FUNCTION_BLOCK "FB_Robot"
{ S7_Optimized_Access := 'TRUE' }
VERSION : 0.1
   VAR
      cmdStatus { S7_SetPoint := 'False'} : "UDT_CMD";
   END_VAR
   VAR RETAIN
      Dispatcher : Array[0..31] of Int;
   END_VAR
   VAR
      Auto : Bool;
      RemoteMode : Bool := TRUE;
      Status : Int;
      oldStatus { ExternalAccessible := 'False'; ExternalVisible := 'False'; ExternalWritable := 'False'} : Int;
      workCondition : Int;   // Status REMOTE, LOCAL, MANUAL
   END_VAR
   VAR RETAIN
      communication_OK : Bool;   // Communication with robot's brain OK
   END_VAR
   VAR
      MissionCode : Int;
      BoxRequested : Int := 1;   // Which warehouse used for mission
      GripperRequested : Int;
      MCRequested : Int;
      PalletRequested : Int;
      Tray_ID : Int;
      Error : Int;   // Every error raised during the cycle
      timeoutLifeBit {InstructionName := 'TON_TIME'; LibVersion := '1.0'; S7_SetPoint := 'False'} : TON_TIME;
   END_VAR
   VAR RETAIN
      Gripper_ID : Array[1..2] of Int;   // Codes of gripper mounted
      GripperOccuped : Array[1..2] of Bool;   // Gripper occuped status
   END_VAR
   VAR
      queryTemp : String;
      paramsTemp { ExternalAccessible := 'False'; ExternalVisible := 'False'; ExternalWritable := 'False'} : Array[0..5] of Int;
      queryStartExecution { ExternalAccessible := 'False'; ExternalVisible := 'False'; ExternalWritable := 'False'} : Bool;
      PollingDB {InstructionName := 'TON_TIME'; LibVersion := '1.0'; S7_SetPoint := 'False'} : Array[1..5] of TON_TIME;
      lastMission { S7_SetPoint := 'True'} : Int;
      WAIT_END_MISSION : Bool;
      HOLD : Bool;
      PalletPosition : Int;
      checkInconsistenceFailed : Bool;
      speedRequest : Int;
      tonCoerenza {InstructionName := 'TON_TIME'; LibVersion := '1.0'; S7_SetPoint := 'False'} : TON_TIME;
      auxOK_old { S7_SetPoint := 'True'} : Bool;
      swapDataReady : Bool;
      tonSwapA {InstructionName := 'TON_TIME'; LibVersion := '1.0'; S7_SetPoint := 'False'} : TON_TIME;
      tonSwapB {InstructionName := 'TON_TIME'; LibVersion := '1.0'} : TON_TIME;
      currentGripperHasHook { S7_SetPoint := 'True'} : Bool;
      PartSubPos : Int;
      declGripper : Int;
      declCont1 : Int;
      declId1 : Int;
      declCont2 : Int;
      declId2 : Int;
      declMap : Int;
      mounted_old : Int := -1;
      closed1_old : Int := -1;
      tonSafetyPub {InstructionName := 'TON_TIME'; LibVersion := '1.0'; S7_SetPoint := 'False'} : TON_TIME;
      zPlaceTemp { S7_SetPoint := 'True'} : DInt;
      PartSubPosMC : Int;
      TrayIdMC : Int;
      xPushTemp : DInt;
      xStopTemp : DInt;
      xPushOffsetMC : DInt;
      xPlaceTemp : DInt;
      declSubPos : Int;
      declStato : Int;
      declTipo : Int;
      retryPick : Bool;
      tonExtract {InstructionName := 'TON_TIME'; LibVersion := '1.0'; S7_SetPoint := 'False'} : TON_TIME;
      OrderIdMC { S7_SetPoint := 'True'} : Int;
      holdButton : Bool;
   END_VAR

   VAR_TEMP
      pieceReq : Int;
      Dispatcher_old : Array[0..31] of Int;
      i : Int;
      RESET_ALL_DISPATCH : Bool;
      temp : Int;
      robotInPendant : Bool;
   END_VAR


BEGIN
	(* Implementato dentro alla classe del Robot
	REGION LIFE BIT
	    "DB_RobotMission".SystemSignals_IN.LIFEBIT_IN := NOT "DB_RobotMissionStatus".systemsignals.LIFE_BIT;

	    #timeoutLifeBit(IN := "DB_RobotMission".SystemSignals_IN.LIFEBIT_IN <> "DB_RobotMissionStatus".systemsignals.LIFE_BIT,
	                    PT := T#3S);

	    IF (#timeoutLifeBit.Q) THEN
	        //salva su DB errore di comunicazione con robot
	        #communication_OK := FALSE;
	    END_IF;
	END_REGION
	*)
	// Il flag va abbassato SOLO quando la query e' entrata davvero nel ponte.
	// Senza il controllo di lunghezza, due stringhe vuote si confermano a vicenda
	// e il flag cade su una query mai partita: la catena resta appesa per sempre
	// (visto 4/9 sulla missione 16, errore 13599 in loop).
	IF LEN(#queryTemp) > 0
	    AND #queryTemp = "SqlCommands".sqlCommands[0]
	    AND #queryStartExecution
	THEN
	    #queryStartExecution := FALSE;
	END_IF;

	REGION Status

	    #Status := DINT_TO_INT("AUTO");
	    IF NOT #HOLD AND ("DB_RobotMissionStatus".StatusCode = "cmd_acquired" OR
	        "DB_RobotMissionStatus".StatusCode = "cmd_executing") THEN
	        #Status := DINT_TO_INT("WORKING");
	    ELSIF NOT #HOLD AND ("DB_RobotMissionStatus".StatusCode = "cmd_aborted" OR
	        "DB_RobotMissionStatus".StatusCode = "cmd_rejected") THEN
	        #Status := DINT_TO_INT("ABORTED");
	    ELSIF NOT #HOLD AND (#Dispatcher["_master"] = 9999 OR
	        #Error <> 0 OR
	        "DB_RobotMissionStatus".StatusRegister.Alarm) THEN
	        #Status := DINT_TO_INT("ALARM");
	    ELSIF NOT #communication_OK THEN
	        #Status := DINT_TO_INT("NOT_DEFINED");
	    ELSIF NOT #HOLD AND NOT "DB_RobotMissionStatus".StatusRegister.Executing AND #Auto THEN
	        #Status := DINT_TO_INT("OFF");
	    ELSIF #HOLD THEN
	        #Status := DINT_TO_INT("HOLD");
	    ELSIF NOT #Auto THEN
	        #Status := DINT_TO_INT("MANUAL");
	    ELSE
	        #Status := DINT_TO_INT("REMOTE");
	    END_IF;

	    IF (#Status <> #oldStatus AND #Status >= 0) THEN
	        IF "DB_RobotMissionStatus".StatusRegister.Alarm THEN
	            "FC_MQTT"(insert := true,
	                      send := false,
	                      topic := 'FROM_PLANT/DESCR/ROBOT',
	                      payload := STRING_TO_WSTRING("INT_TO_STRING_WITHOUT_SIGN"("Alarmcode")));
	        ELSE
	            "FC_MQTT"(insert := true,
	                      "send" := false,
	                      topic := 'FROM_PLANT/DESCR/ROBOT',
	                      payload := STRING_TO_WSTRING("INT_TO_STRING_WITHOUT_SIGN"(#Error)));
	        END_IF;
	        "FC_MQTT"(insert := true,
	                  send := false,
	                  topic := 'FROM_PLANT/STATUS/ROBOT',
	                  payload := STRING_TO_WSTRING("INT_TO_STRING_WITHOUT_SIGN"(#Status)));
	        #oldStatus := #Status;
	    END_IF;

	    //controllo ad ogni ciclo
	    #Status := DINT_TO_INT("REMOTE");

	    IF (#Status <> #workCondition AND #Status >= 0) THEN
	        "FC_MQTT"(insert := true,
	                  send := false,
	                  topic := 'FROM_PLANT/STATUS/ROBOT',
	                  payload := STRING_TO_WSTRING("INT_TO_STRING_WITHOUT_SIGN"(#Status)));
	        #workCondition := #Status;
	    END_IF;
	END_REGION ;

	FOR #i := 0 TO 31 DO
	    #Dispatcher_old[#i] := #Dispatcher[#i];
	END_FOR;

	REGION Manager CMD from HMI
	    // Modo cella: DB_Robot.RemoteMode (TRUE = automatico, FALSE = manuale/locale).
	    // Scritto SOLO qui dai comandi 81/82 — il robot non partecipa al giro modalita'.
	    // Robot sotto pendant (manuale suo): nessun comando di movimento accettato.
	    #robotInPendant := "sys_manual_T1" OR "sys_manual_Full";
	    #RemoteMode := NOT #HOLD;   // modo cella derivato: HOLD = manuale

	    // ---- Comandi accettati in ogni condizione ----
	    IF "DB_MQTT".lastTopicReceived = 'ROBOT' THEN
	        CASE "DB_MQTT".lastCmdReceived OF
	            "CMD_HOLD":
	                // IL PULSANTE E' MASTER (19/9): un hold messo col pulsante fisico
	                // lo toglie solo il pulsante. Dal pannello si puo' mettere
	                // l'hold e togliere il proprio, non quello di chi sta in campo
	                // davanti alla cella. La gerarchia la tiene FB5, che scrive
	                // holdButton: qui si legge e basta.
	                IF NOT #holdButton THEN
	                    #HOLD := NOT #HOLD;
	                END_IF;
	            "CMD_changeRobotSpeed":
	                #speedRequest := "DB_MQTT".lastParams[0];
	            "CMD_Refresh":  // 90: ripubblica tutti gli one-shot
	                #oldStatus := -1;
	                #lastMission := -1;
	                #auxOK_old := NOT "Main_Safety_RTG1_DB".Aux_OK;
	                #mounted_old := -1;
	                #closed1_old := -1;
	                "DB_MC1".brandID_req_old := -1;
	                "DB_MC1".brandID_act_old := -1;
	                "DB_MC1".declPallet_old := -1;
	                "DB_MC1".declPiece_old := -1;
	                "DB_MC1".declVice_old := -1;
	                FOR #i := 0 TO 31 DO
	                    #Dispatcher_old[#i] := -1;
	                END_FOR;
	                "DB_MQTT".lastCmdReceived := 0;
	        END_CASE;
	    END_IF;

	    // ---- Restart main program: solo con orchestrazione in HOLD ----
	    IF "DB_MQTT".lastTopicReceived = 'ROBOT' AND #HOLD THEN
	        CASE "DB_MQTT".lastCmdReceived OF
	            "CMD_RestartMainProg":
	                "DB_RobotMission".Command := "CMD_RestartMainProg";
	                "DB_MQTT".lastCmdReceived := 0;
	                #WAIT_END_MISSION := FALSE;
	                // il restart del programma robot abbandona la missione in corso (5/10):
	                // si azzerano le catene come per i movimenti manuali, altrimenti
	                // restano ad aspettare un "eseguito" che non arrivera' mai.
	                #RESET_ALL_DISPATCH := TRUE;
	                #MissionCode := 0;
	        END_CASE;
	    END_IF;

	    // ---- Canale libero: modo cella + reset, validi in ENTRAMBI i modi ----
	    IF "DB_MQTT".lastTopicReceived = 'ROBOT'
	        AND "DB_RobotMissionStatus".StatusCode <> "cmd_acquired"
	        AND "DB_RobotMissionStatus".StatusCode <> "cmd_executing"
	    THEN
	        CASE "DB_MQTT".lastCmdReceived OF
	            "CMD_RobotReset":
	                #Error := 0;
	                "DB_RobotMission".Command := "CMD_RobotReset"; //arriva direttamente nella missione robot
	                #MissionCode := 0;
	                #RESET_ALL_DISPATCH := TRUE;
	                #WAIT_END_MISSION := TRUE;

	                // IL RESET DEVE FERMARE ANCHE L'ORCHESTRAZIONE MACCHINA (16/9).
	                // Prima azzerava solo le catene di FB7: FB204 restava dov'era e
	                // riprendeva da uno stato che non esisteva piu'. Visto in campo:
	                // reset a meta' deposito del finito -> il 95 substate 1 vede
	                // MissionCode = 0 (appena azzerato QUI) e conclude che lo scarico
	                // e' finito, prosegue sui registri di bordo troncati, e arriva a
	                // rilanciare la RICETTA su un pezzo GIA' LAVORATO ancora in morsa.
	                "DB_MC1".Dispatcher["_master"] := 0;
	                "DB_MC2".Dispatcher["_master"] := 0;

	                "DB_MQTT".lastCmdReceived := 0;
	        END_CASE;

	        // ---- Comandi manuali: SOLO cella in locale E robot non in pendant ----
	        IF NOT #RemoteMode AND NOT #robotInPendant THEN
	            CASE "DB_MQTT".lastCmdReceived OF
	                "CMD_RobotToHomePos":
	                    "DB_RobotMission".Command := "CMD_RobotToHomePos";
	                    "DB_MQTT".lastCmdReceived := 0;
	                    #WAIT_END_MISSION := TRUE;
	                    #RESET_ALL_DISPATCH := TRUE; // abort missioni pendenti: no falso latch da 3 del movimento manuale
	                    #MissionCode := 0;
	                "CMD_RobotMaintenancePos":
	                    "DB_RobotMission".Command := "CMD_RobotMaintenancePos";
	                    "DB_MQTT".lastCmdReceived := 0;
	                    #WAIT_END_MISSION := TRUE;
	                    #RESET_ALL_DISPATCH := TRUE; // abort missioni pendenti: no falso latch da 3 del movimento manuale
	                    #MissionCode := 0;
	                "CMD_RobotPositioning":
	                    "DB_RobotMission".Command := "CMD_RobotPositioning"; // riceve comandi del tipo 15;1
	                    "DB_RobotMission".Unit_code := "DB_MQTT".lastParams[0];
	                    "DB_MQTT".lastCmdReceived := 0;
	                    #WAIT_END_MISSION := TRUE;
	                    #RESET_ALL_DISPATCH := TRUE; // abort missioni pendenti: no falso latch da 3 del movimento manuale
	                    #MissionCode := 0;
	                "CMD_RobotPositioning_BOX1":
	                    "DB_RobotMission".Command := "CMD_RobotPositioning";
	                    "DB_RobotMission".Unit_code := "Warehouse1";
	                    "DB_MQTT".lastCmdReceived := 0;
	                    #WAIT_END_MISSION := TRUE;
	                    #RESET_ALL_DISPATCH := TRUE; // abort missioni pendenti: no falso latch da 3 del movimento manuale
	                    #MissionCode := 0;
	                "CMD_RobotPositioning_MC1":
	                    "DB_RobotMission".Command := "CMD_RobotPositioning";
	                    "DB_RobotMission".Unit_code := "MC1";
	                    "DB_MQTT".lastCmdReceived := 0;
	                    #WAIT_END_MISSION := TRUE;
	                    #RESET_ALL_DISPATCH := TRUE; // abort missioni pendenti: no falso latch da 3 del movimento manuale
	                    #MissionCode := 0;
	                "CMD_RobotPickGripper":
	                    "DB_MQTT".lastCmdReceived := 0;
	                    #MissionCode := "MISSION_LoadGripper";
	                    #GripperRequested := "DB_MQTT".lastParams[0];
	                    #WAIT_END_MISSION := TRUE;
	                "CMD_RobotRemoveGripper":
	                    "DB_MQTT".lastCmdReceived := 0;
	                    #MissionCode := "MISSION_UnloadGripper";
	                    #WAIT_END_MISSION := TRUE;
	                "CMD_RobotExtractTray":
	                    #Tray_ID := DINT_TO_INT("DB_MQTT".lastParams[0]);  // <-- riga nuova
	                    #MissionCode := "MISSION_ExtractTray";
	                    "DB_MQTT".lastCmdReceived := 0;
	                    #WAIT_END_MISSION := TRUE;
	                "CMD_RobotReleaseTray":
	                    #MissionCode := "MISSION_ReleaseTray";
	                    "DB_MQTT".lastCmdReceived := 0;
	                    #WAIT_END_MISSION := TRUE;
	                "CMD_RobotPickObject":
	                    "DB_RobotMission".Object_Type := "DB_MQTT".lastParams[0];
	                    #PalletRequested := "DB_MQTT".lastParams[1];
	                    CASE "DB_RobotMission".Object_Type OF
	                        "Pallet":
	                            #PalletPosition := "DB_MQTT".lastParams[2];
	                            IF #PalletPosition = 0 THEN
	                                #MissionCode := "MISSION_PickPallet_MC_HMI";
	                                #MCRequested := 1;
	                            ELSE
	                                #MissionCode := "MISSION_Load_Pallet";
	                                #MCRequested := 0;
	                            END_IF;
	                            "DB_MQTT".lastCmdReceived := 0;
	                            #WAIT_END_MISSION := TRUE;
	                        "Part": //TODO
	                            ;
	                        "ViceWithoutPart":
	                            ;
	                        "ViceWithPart":
	                            ;
	                    END_CASE;
	                "CMD_RobotPlaceObject":
	                    "DB_RobotMission".Object_Type := "DB_MQTT".lastParams[0];
	                    #PalletRequested := "DB_MQTT".lastParams[1];
	                    CASE "DB_RobotMission".Object_Type OF
	                        "Pallet":
	                            #PalletPosition := "DB_MQTT".lastParams[2];
	                            IF #PalletPosition = 0 THEN
	                                #MissionCode := "MISSION_PlacePallet_MC_HMI";
	                                #MCRequested := 1;
	                            ELSE
	                                #MissionCode := "MISSION_Unload_Pallet";
	                                #MCRequested := 0;
	                            END_IF;
	                            "DB_MQTT".lastCmdReceived := 0;
	                            #WAIT_END_MISSION := TRUE;
	                        "Part": //TODO
	                            ;
	                        "ViceWithoutPart":
	                            ;
	                        "ViceWithPart":
	                            ;
	                    END_CASE;
	                "CMD_HMI_SwapGripper":
	                    "DB_MQTT".lastCmdReceived := 0;
	                    #GripperRequested := "DB_MQTT".lastParams[0];
	                    #MissionCode := "MISSION_SwapGripper";
	                    #WAIT_END_MISSION := TRUE;

	                "CMD_DeclarePosition_TRAY":   // 39;subpos;stato  (2 vuota, 4 grezzo, 5 finito)
	                    #declSubPos := DINT_TO_INT("DB_MQTT".lastParams[0]);
	                    #declStato := DINT_TO_INT("DB_MQTT".lastParams[1]);
	                    #declTipo := 0;                         // ramo STATO, non TIPO
	                    IF "DB_BOX_1".ExtractedTray <= 0 THEN
	                        #Error := 20001;                    // nessun cassetto estratto
	                    ELSIF #declSubPos <= 0 THEN
	                        #Error := 20002;                    // posizione non valida
	                    ELSIF #declStato <> 2 AND #declStato <> 4 AND #declStato <> 5 THEN
	                        #Error := 20005;                    // stato non ammesso
	                    ELSE
	                        #Dispatcher["_Declare_Position"] := 10;
	                    END_IF;
	                    "DB_MQTT".lastCmdReceived := 0;
	                    #WAIT_END_MISSION := FALSE;   // nessun movimento robot

	                "CMD_DeclarePieceType_TRAY":   // 44;partType  tipo pezzo dell'INTERO cassetto estratto
	                    #declTipo := DINT_TO_INT("DB_MQTT".lastParams[0]);
	                    IF "DB_BOX_1".ExtractedTray <= 0 THEN
	                        #Error := 20001;                    // nessun cassetto estratto
	                    ELSIF #declTipo <= 0 THEN
	                        #Error := 20008;                    // tipo pezzo non valido
	                    ELSE
	                        #Dispatcher["_Declare_Position"] := 15;   // ramo TIPO
	                    END_IF;
	                    "DB_MQTT".lastCmdReceived := 0;
	                    #WAIT_END_MISSION := FALSE;   // nessun movimento robot

	                "CMD_RobotPickPartTray":   // 27;subpos;gripperID  (gripperID 0 = pinza a bordo)
	                    IF "DB_BOX_1".ExtractedTray <= 0 THEN
	                        #Error := 20001;                    // nessun cassetto estratto
	                    ELSIF DINT_TO_INT("DB_MQTT".lastParams[0]) <= 0 THEN
	                        #Error := 20002;                    // posizione pezzo non valida
	                    ELSIF DINT_TO_INT("DB_MQTT".lastParams[1]) = 0 AND #Gripper_ID[1] = 0 THEN
	                        #Error := 22;                       // flangia vuota e nessuna pinza richiesta
	                    ELSE
	                        #PartSubPos := DINT_TO_INT("DB_MQTT".lastParams[0]);
	                        #GripperRequested := DINT_TO_INT("DB_MQTT".lastParams[1]);
	                        IF #GripperRequested = 0 THEN
	                            #GripperRequested := #Gripper_ID[1];
	                        END_IF;
	                        #Tray_ID := "DB_BOX_1".ExtractedTray;
	                        #MCRequested := 0;
	                        #MissionCode := "MISSION_PickPart_TRAY_HMI";
	                        #WAIT_END_MISSION := TRUE;
	                    END_IF;
	                    "DB_MQTT".lastCmdReceived := 0;

	                "CMD_RobotPlacePartTray":  // 28;subpos  (0 = prima posizione vuota)
	                    IF "DB_BOX_1".ExtractedTray <= 0 THEN
	                        #Error := 20001;
	                    ELSE
	                        #PartSubPos := DINT_TO_INT("DB_MQTT".lastParams[0]);
	                        #Tray_ID := "DB_BOX_1".ExtractedTray;
	                        #MCRequested := 0;
	                        #MissionCode := "MISSION_PlacePart_TRAY_HMI";
	                        #WAIT_END_MISSION := TRUE;
	                    END_IF;
	                    "DB_MQTT".lastCmdReceived := 0;

	                "CMD_RobotPickPartMC":     // 29;gripperID  (0 = pinza a bordo)
	                    IF DINT_TO_INT("DB_MQTT".lastParams[0]) = 0 AND #Gripper_ID[1] = 0 THEN
	                        #Error := 22;
	                    ELSE
	                        #GripperRequested := DINT_TO_INT("DB_MQTT".lastParams[0]);
	                        IF #GripperRequested = 0 THEN
	                            #GripperRequested := #Gripper_ID[1];
	                        END_IF;
	                        #MCRequested := 1;                  // MC2 non esiste in questa cella
	                        #MissionCode := "MISSION_PickPart_MC_HMI";
	                        #WAIT_END_MISSION := TRUE;
	                    END_IF;
	                    "DB_MQTT".lastCmdReceived := 0;

	                "CMD_RobotPlacePartMC":    // 30  (pezzo a bordo -> morsa MC1)
	                    #MCRequested := 1;
	                    #GripperRequested := #Gripper_ID[1];
	                    #MissionCode := "MISSION_PlacePart_MC_HMI";
	                    #WAIT_END_MISSION := TRUE;
	                    "DB_MQTT".lastCmdReceived := 0;
	                "CMD_RobotPickPlacePartMC":  // 244  (finito da morsa + grezzo in morsa, un ingresso)
	                    IF NOT #GripperOccuped[1] THEN
	                        #Error := 20003;                    // nessun grezzo a bordo lato 1
	                    ELSIF #GripperOccuped[2] THEN
	                        #Error := 20004;                    // lato finito gia' occupato
	                    ELSE
	                        #MCRequested := 1;
	                        #GripperRequested := #Gripper_ID[1];
	                        #MissionCode := "MISSION_PickPlacePart_MC";
	                        #WAIT_END_MISSION := TRUE;
	                    END_IF;
	                    "DB_MQTT".lastCmdReceived := 0;
	                "CMD_OpenGripper1":
	                    "DB_MQTT".lastCmdReceived := 0;
	                    #MissionCode := "MISSION_OpenGripper1";
	                    #WAIT_END_MISSION := TRUE;
	                "CMD_CloseGripper1":
	                    "DB_MQTT".lastCmdReceived := 0;
	                    #MissionCode := "MISSION_CloseGripper1";
	                    #WAIT_END_MISSION := TRUE;
	                "CMD_OpenGripper2":
	                    IF #Gripper_ID[2] = 0 THEN
	                        #Error := 944;   // lato 2 inesistente sulla pinza a bordo
	                    ELSE
	                        #MissionCode := "MISSION_OpenGripper2";
	                        #WAIT_END_MISSION := TRUE;
	                    END_IF;
	                    "DB_MQTT".lastCmdReceived := 0;
	                "CMD_CloseGripper2":
	                    IF #Gripper_ID[2] = 0 THEN
	                        #Error := 944;
	                    ELSE
	                        #MissionCode := "MISSION_CloseGripper2";
	                        #WAIT_END_MISSION := TRUE;
	                    END_IF;
	                    "DB_MQTT".lastCmdReceived := 0;
	                "CMD_RobotDeclareState":   // 35;gripperID;cont1;id1;cont2;id2  (cont: 0=vuoto 1=grezzo 2=finito 3=pallet)
	                    #declGripper := DINT_TO_INT("DB_MQTT".lastParams[0]);
	                    #declCont1 := DINT_TO_INT("DB_MQTT".lastParams[1]);
	                    #declId1 := DINT_TO_INT("DB_MQTT".lastParams[2]);
	                    #declCont2 := DINT_TO_INT("DB_MQTT".lastParams[3]);
	                    #declId2 := DINT_TO_INT("DB_MQTT".lastParams[4]);
	                    #Error := 0;
	                    #MissionCode := 0;
	                    #Dispatcher["_Declare_State"] := 10;
	                    "DB_MQTT".lastCmdReceived := 0;
	                    #WAIT_END_MISSION := FALSE;   // nessun movimento robot
	            END_CASE;
	        END_IF;
	    END_IF;

	    // ---- Completamento comando (invariato) ----
	    IF #WAIT_END_MISSION THEN
	        IF "DB_RobotMissionStatus".StatusCode = "cmd_executed" THEN
	            #WAIT_END_MISSION := FALSE;
	            //sync with robot
	            "DB_RobotMission".Command := 0;
	        ELSIF "DB_RobotMissionStatus".StatusCode = "cmd_rejected" OR "DB_RobotMissionStatus".StatusCode = "cmd_aborted" THEN
	            #WAIT_END_MISSION := FALSE;
	            // COMANDO MANUALE RIFIUTATO O ABORTITO (5/10): senza missione in
	            // corso si azzera anche il comando. Altrimenti il 4/5 resta esposto
	            // e la sorveglianza qui sotto lo attribuirebbe alla missione dopo.
	            IF #Dispatcher["_master"] = 0 THEN
	                "DB_RobotMission".Command := 0;
	            END_IF;
	        END_IF;
	    END_IF;

	    // ---- Sorveglianza risposta robot (5/10) ----
	    // Le risposte 4 (abortito) e 5 (rifiutato) erano gestite solo qui sopra,
	    // per i comandi manuali, e nelle catene chele. Le catene pezzi e cassetto
	    // restavano ad aspettare un 3 che non arriva: cella ferma con Error = 0 e
	    // nessuna spiegazione. Con una missione in corso e un comando al robot,
	    // una risposta anomala che dura 1 s diventa un errore dichiarato, che il
	    // reset (99) toglie. Il secondo di filtro evita di leggere lo StatusCode
	    // rimasto dal comando precedente nei primi cicli dopo un comando nuovo.
	    // Esclusi: lo scan del reset (99, AUX, ResetAreaRobot), in cui il master
	    // e' ancora valorizzato; l'HOLD, in cui il programma robot e' in pausa; la
	    // ripartenza del programma dopo HOLD o restart (FB8 dispatcher 0 e 1), che
	    // puo' durare fino a 17 s.
	    // Il codice 6 ("interrotto") NON e' gestito: non e' fra le costanti cmd_
	    // e va prima confermato col robotista.
	    // PollingDB[1] e' un timer gia' dichiarato e mai usato: nessuna variabile
	    // nuova, interfaccia invariata.
	    #PollingDB[1](IN := #Dispatcher["_master"] <> 0
	                  AND #Error = 0
	                  AND "DB_RobotMission".Command <> 0
	                  AND NOT #HOLD
	                  AND NOT #RESET_ALL_DISPATCH
	                  AND NOT "Start_AUX"
	                  AND NOT "ResetAreaRobot"
	                  AND "DB_Robot_Efort".dispatcher[0] = 0
	                  AND "DB_Robot_Efort".dispatcher[1] = 0
	                  AND ("DB_RobotMissionStatus".StatusCode = "cmd_aborted"
	                  OR "DB_RobotMissionStatus".StatusCode = "cmd_rejected"),
	                  PT := T#1s);
	    IF #PollingDB[1].Q THEN
	        IF "DB_RobotMissionStatus".StatusCode = "cmd_aborted" THEN
	            #Error := 961;   // missione abortita dal robot
	        ELSE
	            #Error := 962;   // comando rifiutato dal robot
	        END_IF;
	    END_IF;
	END_REGION

	REGION Cycle MASTER ROBOT

	    //DA TESTARE
	    (*IF "DB_RobotMissionStatus".StatusCode = "cmd_executed" THEN
	        "DB_RobotMission".Command := 0;
	    END_IF;
	    *)

	    IF NOT "Main_Safety_RTG1_DB".Aux_OK THEN
	        #MissionCode := 0;
	    END_IF;

	    #tonSwapA(IN := #Dispatcher["_master"] >= 973 AND #Dispatcher["_master"] <= 974,
	              PT := T#60s);
	    // TIMEOUT ESTESO AL 9781 (17/9): il 978 ora chiude in un ciclo e passa la
	    // registrazione alla catena unica. Senza estendere la sorveglianza, un ponte
	    // SQL occupato lascerebbe il master appeso al 9781 in silenzio, con la pinza
	    // gia' a bordo.
	    #tonSwapB(IN := #Dispatcher["_master"] = 978 OR #Dispatcher["_master"] = 9781,
	              PT := T#60s);
	    IF (#tonSwapA.Q OR #tonSwapB.Q) AND #Error = 0 THEN
	        #Error := 943;  // swap: timeout di fase (deposito o prelievo)
	    END_IF;

	    // SORVEGLIANZA CATENA CASSETTO (18/9): e' la terza catena che si pianta in
	    // silenzio. Il 12 aveva un ramo mancante — corretto — ma il principio resta:
	    // una catena senza timeout, quando si ferma, ferma anche il 750 che la
	    // aspetta e il 58 di FB204 che aspetta il 750, e nessuno lo dice.
	    // Tre minuti coprono estrazione e rilascio con margine largo.
	    #tonExtract(IN := #Dispatcher["Extract_TRAY"] > 0 OR #Dispatcher["Release_TRAY"] > 0,
	                PT := T#180s);
	    IF #tonExtract.Q AND #Error = 0 THEN
	        #Error := 19003;   // catena cassetto: timeout
	    END_IF;

	    IF #communication_OK THEN
	        CASE #Dispatcher["_master"] OF
	            0:
	                CASE #MissionCode OF
	                    "MISSION_LoadPallet_MC":        // pallet: Robot -> MC
	                        IF #RemoteMode AND
	                            "DB_RobotMissionStatus".StatusCode = "cmd_waitingNewCmd"
	                        THEN
	                            IF #MCRequested = 1 THEN
	                                IF "DB_MC1".order.GRIPPER4PALLET > 0 THEN
	                                    #GripperRequested := DINT_TO_INT("DB_MC1".order.GRIPPER4PALLET);
	                                    #Dispatcher["_master"] := 100;
	                                END_IF;
	                            ELSIF #MCRequested = 2 THEN
	                                IF "DB_MC1".order.GRIPPER4PALLET > 0 THEN
	                                    #GripperRequested := DINT_TO_INT("DB_MC2".order.GRIPPER4PALLET);
	                                    #Dispatcher["_master"] := 100;
	                                END_IF;
	                            ELSE
	                                #Dispatcher["_master"] := 0;
	                            END_IF;
	                        END_IF;
	                    "MISSION_UnloadPallet_MC":      // pallet: MC -> Robot
	                        IF #RemoteMode AND
	                            "DB_RobotMissionStatus".StatusCode = "cmd_waitingNewCmd"
	                        THEN
	                            IF #MCRequested = 1 THEN
	                                #GripperRequested := DINT_TO_INT("DB_MC1".order.GRIPPER4PALLET);
	                            ELSE
	                                #GripperRequested := DINT_TO_INT("DB_MC2".order.GRIPPER4PALLET);
	                            END_IF;
	                            #Dispatcher["_master"] := 200;
	                        END_IF;
	                    "MISSION_LoadPart_MC":          // part: Robot -> MC
	                        IF #RemoteMode AND
	                            "DB_RobotMissionStatus".StatusCode = "cmd_waitingNewCmd"
	                        THEN
	                            IF #MCRequested = 1 THEN
	                                #GripperRequested := DINT_TO_INT("DB_MC1".order.GRIPPER);
	                            ELSE
	                                #GripperRequested := DINT_TO_INT("DB_MC2".order.GRIPPER);
	                            END_IF;
	                            IF #GripperRequested > 0 THEN
	                                #Dispatcher["_master"] := 300;
	                            ELSE
	                                #Error := "MISSION_LoadPart_MC" * 100 + 10;  //Error 12010
	                            END_IF;
	                        END_IF;
	                    "MISSION_UnloadPart_MC":        // part: MC -> Robot
	                        IF #RemoteMode AND
	                            "DB_RobotMissionStatus".StatusCode = "cmd_waitingNewCmd"
	                        THEN
	                            IF #MCRequested = 1 THEN
	                                #GripperRequested := DINT_TO_INT("DB_MC1".order.GRIPPER);
	                            ELSE
	                                #GripperRequested := DINT_TO_INT("DB_MC2".order.GRIPPER);
	                            END_IF;
	                            IF #GripperRequested > 0 THEN
	                                #Dispatcher["_master"] := 400;
	                            ELSE
	                                #Error := "MISSION_UnloadPart_MC" * 100 + 10;  //Error 13010
	                            END_IF;
	                        END_IF;
	                    "MISSION_PickPlacePart_MC":     // 16: preleva finito + deposita grezzo, un ingresso solo
	                        IF "DB_RobotMissionStatus".StatusCode = "cmd_waitingNewCmd" AND #Error = 0 THEN
	                            IF #GripperRequested > 0 THEN
	                                #Dispatcher["_master"] := 1400;
	                            ELSE
	                                #Error := "MISSION_PickPlacePart_MC" * 100 + 10;
	                            END_IF;
	                        END_IF;
	                    "MISSION_LoadPartOnRobot":      // part: TRAY -> Robot
	                        IF #RemoteMode AND
	                            "DB_RobotMissionStatus".StatusCode = "cmd_waitingNewCmd"
	                        THEN
	                            IF #MCRequested = 1 THEN
	                                #GripperRequested := DINT_TO_INT("DB_MC1".order.GRIPPER);
	                            ELSIF #MCRequested = 2 THEN
	                                #GripperRequested := DINT_TO_INT("DB_MC2".order.GRIPPER);
	                            ELSE
	                                #GripperRequested := #Gripper_ID[1];   // nessuna MC indicata: pinza a bordo
	                            END_IF;
	                            IF #GripperRequested > 0 THEN
	                                #Dispatcher["_master"] := 500;
	                            ELSE
	                                #Error := "MISSION_LoadPartOnRobot" * 100 + 10;
	                            END_IF;
	                        END_IF;
	                    "MISSION_UnloadPartFromRobot":  // part: Robot -> TRAY
	                        IF #RemoteMode AND
	                            "DB_RobotMissionStatus".StatusCode = "cmd_waitingNewCmd"
	                        THEN
	                            #Dispatcher["_master"] := 600;
	                            // IF #MCRequested = 1 THEN
	                            //     #GripperRequested := DINT_TO_INT("DB_MC1".order.GRIPPER);
	                            //     #Dispatcher["_master"] := 600;
	                            // ELSE
	                            //     #GripperRequested := DINT_TO_INT("DB_MC2".order.GRIPPER);
	                            //     #Dispatcher["_master"] := 600;
	                            // END_IF;
	                        END_IF;

	                        // COMMANDS NOT NEEDS RemoteMode ACTIVE

	                    "MISSION_ExtractTray":
	                        //devo prima mandare dentro gli altri se ci sono?
	                        IF #Dispatcher["Extract_TRAY"] = 0 AND #Error = 0 THEN
	                            #Dispatcher["_master"] := 700;
	                        END_IF;
	                    "MISSION_ReleaseTray":
	                        IF #Dispatcher["Release_TRAY"] = 0 AND #Error = 0 THEN
	                            IF "DB_BOX_1".ExtractedTray > 0 THEN
	                                #Dispatcher["Release_TRAY"] := 10;
	                                #Dispatcher["_master"] := 800;
	                            ELSE
	                                #MissionCode := 0;
	                                #Dispatcher["_master"] := 0;
	                            END_IF;
	                        END_IF;
	                    "MISSION_UnloadGripper":
	                        IF #Gripper_ID[1] > 0 AND #Dispatcher["_Gripper_Robot_to_TRAY"] = 0 THEN
	                            #Dispatcher["_Gripper_Robot_to_TRAY"] := 10;
	                            #Dispatcher["_master"] := 900;
	                        ELSIF #Gripper_ID[1] <= 0 THEN
	                            #Error := 936;  // scarico richiesto ma nessuna pinza registrata al sistema
	                        END_IF;
	                    "MISSION_LoadGripper":
	                        IF "Gripper_mounted" THEN
	                            #Error := 935;
	                        ELSE
	                            #Dispatcher["_Gripper_TRAY_to_Robot"] := 10;
	                            #MCRequested := 0;

	                            #Dispatcher["_master"] := 950;
	                        END_IF;
	                    "MISSION_SwapGripper":
	                        IF #GripperRequested <= 0 THEN
	                            #Error := 937;          // swap: pinza target non valida
	                            #MissionCode := 0;
	                        ELSIF #GripperRequested = #Gripper_ID[1] THEN
	                            #Error := 939;          // swap: pinza richiesta gia' a bordo
	                            #MissionCode := 0;
	                        ELSIF #Gripper_ID[1] = 0 THEN
	                            // flangia vuota: degenera nel carico classico (chiude via 950/960)
	                            #Dispatcher["_Gripper_TRAY_to_Robot"] := 10;
	                            #MCRequested := 0;
	                            #Dispatcher["_master"] := 950;
	                        ELSE
	                            #swapDataReady := FALSE;
	                            #Dispatcher["_master"] := 970;
	                        END_IF;
	                    "MISSION_LoadManVice":
	                        ; //TODO
	                    "MISSION_UnloadManVice":
	                        ; //TODO
	                    "MISSION_Unload_Pallet":
	                        IF NOT #RemoteMode THEN
	                            IF #MCRequested = 0 THEN
	                                #Dispatcher["_master"] := 1500;
	                            END_IF;
	                        END_IF;  //TODO
	                    "MISSION_Load_Pallet":                 // pick Object -> Robot (HMI command)
	                        IF NOT #RemoteMode THEN
	                            IF #MCRequested = 0 THEN
	                                #Dispatcher["_master"] := 1000;
	                            END_IF;
	                        END_IF;

	                    "MISSION_PickPart_TRAY_HMI":
	                        IF NOT #RemoteMode AND #Error = 0 THEN
	                            #Dispatcher["_master"] := 1100;
	                        END_IF;
	                    "MISSION_PlacePart_TRAY_HMI":
	                        IF NOT #RemoteMode AND #Error = 0 THEN
	                            #Dispatcher["_Part_Robot_to_TRAY"] := 10;
	                            #Dispatcher["_master"] := 1150;
	                        END_IF;
	                    "MISSION_PickPart_MC_HMI":
	                        IF NOT #RemoteMode AND #Error = 0 THEN
	                            #Dispatcher["_master"] := 1200;
	                        END_IF;
	                    "MISSION_PlacePart_MC_HMI":
	                        IF NOT #RemoteMode AND #Error = 0 THEN
	                            #Dispatcher["_Part_Robot_to_MC"] := 10;
	                            #Dispatcher["_master"] := 1250;
	                        END_IF;
	                    "MISSION_PickPallet_MC_HMI":
	                        IF NOT #RemoteMode AND #Error = 0 THEN
	                            #Dispatcher["_master"] := 1300;
	                        END_IF;
	                    "MISSION_PlacePallet_MC_HMI":
	                        IF NOT #RemoteMode AND #Error = 0 THEN
	                            #Dispatcher["_Pallet_Robot_to_MC"] := 10;
	                            #Dispatcher["_master"] := 1350;
	                        END_IF;

	                    "MISSION_OpenGripper1":
	                        IF NOT #RemoteMode AND #Error = 0 THEN
	                            #Dispatcher["_master"] := 1600;
	                        END_IF;
	                    "MISSION_CloseGripper1":
	                        IF NOT #RemoteMode AND #Error = 0 THEN
	                            #Dispatcher["_master"] := 1620;
	                        END_IF;
	                    "MISSION_OpenGripper2":
	                        IF NOT #RemoteMode AND #Error = 0 THEN
	                            #Dispatcher["_master"] := 1640;
	                        END_IF;
	                    "MISSION_CloseGripper2":
	                        IF NOT #RemoteMode AND #Error = 0 THEN
	                            #Dispatcher["_master"] := 1660;
	                        END_IF;
	                    "MISSION_PositioningMC_AUTO":   // avvicinamento a MC1 in attesa porta
	                        IF #RemoteMode AND
	                            "DB_RobotMissionStatus".StatusCode = "cmd_waitingNewCmd"
	                        THEN
	                            "DB_RobotMission".Unit_code := "MC1";
	                            "DB_RobotMission".Command := "CMD_RobotPositioning";
	                            #Dispatcher["_master"] := 1700;
	                        END_IF;
	                    "MISSION_RobotHome_AUTO":   // ritorno in home a fine produzione
	                        // CMD_RobotToHomePos e' accettato SOLO in manuale (la
	                        // REGION comandi HMI lo chiude dentro NOT RemoteMode), e
	                        // in automatico non e' raggiungibile. Serviva una missione
	                        // dedicata, sul modello di MISSION_PositioningMC_AUTO che
	                        // esiste per lo stesso identico motivo.
	                        IF #RemoteMode AND
	                            "DB_RobotMissionStatus".StatusCode = "cmd_waitingNewCmd"
	                        THEN
	                            "DB_RobotMission".Command := "CMD_RobotToHomePos";
	                            #Dispatcher["_master"] := 1750;
	                        END_IF;

	                END_CASE;

	                ///////////////////////////
	            100: //MISSION_LoadPallet_MC1 or MC2
	                // TRE RAMI, come il 1100 (17/9): il controllo sulla sola
	                // disuguaglianza lanciava lo scarico anche a FLANGIA NUDA —
	                // Gripper_ID[1]=0 e' diverso da qualunque pinza richiesta, quindi
	                // _Gripper_Robot_to_TRAY partiva e componeva la query con id=0,
	                // che a scaffale non esiste: zero righe, errore 990, master
	                // appeso al 110 per sempre. Visto in campo avviando senza pinza.
	                IF #Gripper_ID[1] <> #GripperRequested AND #Gripper_ID[1] > 0 THEN
	                    #Dispatcher["_Gripper_Robot_to_TRAY"] := 10;
	                    #Dispatcher["_master"] := 110;
	                ELSIF #Gripper_ID[1] = 0 THEN
	                    // flangia nuda: niente da scaricare, si carica e basta
	                    #Dispatcher["_Gripper_TRAY_to_Robot"] := 10;
	                    #Dispatcher["_master"] := 115;
	                ELSE
	                    #Dispatcher["_master"] := 120;
	                END_IF;
	            110:
	                // GUARDIA SULLA CATENA DI SCARICO (16/9): serve anche la conferma
	                // che _Gripper_Robot_to_TRAY abbia CHIUSO, non solo che il registro
	                // sia tornato a zero. Gripper_ID[1] viene azzerato allo stato 40
	                // della catena di scarico, che poi passa al 50 e aspetta l'update
	                // del database: in quella finestra il registro dice gia' "flangia
	                // nuda" mentre la catena sta ancora lavorando, e il carico partiva
	                // sovrapponendosi allo scarico sullo stesso ponte SQL.
	                // Gli altri rami analoghi — 210, 310, 410 — la guardia ce l'hanno
	                // gia': il 110 era l'unico rimasto scoperto.
	                IF #Gripper_ID[1] = 0 AND #Dispatcher["_Gripper_Robot_to_TRAY"] = 0 THEN
	                    #Dispatcher["_Gripper_TRAY_to_Robot"] := 10;
	                    #Dispatcher["_master"] := 115;
	                END_IF;

	            115:
	                IF #Dispatcher["_Gripper_TRAY_to_Robot"] = 0 THEN
	                    #Dispatcher["get_TCP_Data"] := 10;
	                    #Dispatcher["_master"] := 120;
	                END_IF;
	            120: //gripper OK -> start mission
	                // TCP NON AGGIORNATO = NIENTE MISSIONE (5/10): se get_TCP_Data chiude
	                // in errore (2205 pinza assente dal DB, 99 errore DB) il robot ha
	                // ancora il TCP della pinza precedente. Prima si lanciava comunque il
	                // prelievo pallet; ora la missione si chiude e resta l'errore.
	                IF #Dispatcher["get_TCP_Data"] = 0 AND #Error <> 0 THEN
	                    #MissionCode := 0;
	                    #MCRequested := 0;
	                    #Dispatcher["_master"] := 0;
	                ELSIF #Gripper_ID[1] = #GripperRequested AND #Dispatcher["get_TCP_Data"] = 0 THEN
	                    #Dispatcher["_Pallet_TRAY_to_Robot"] := 10;
	                    #Dispatcher["_master"] := 130;
	                END_IF;
	            130:
	                IF #GripperOccuped[1] AND
	                    "DB_RobotMissionStatus".StatusCode = "cmd_waitingNewCmd" AND  //"cmd_executed"   ****
	                    #Dispatcher["_Pallet_TRAY_to_Robot"] = 0 THEN // #Dispatcher["updatePartOnRobot"] = 0 THEN

	                    #Dispatcher["_Pallet_Robot_to_MC"] := 10;
	                    "DB_RobotMission".Command := 0;  ///\\\

	                    #Dispatcher["_master"] := 140;
	                END_IF;
	            140: //Mission ended
	                IF #Dispatcher["_Pallet_Robot_to_MC"] = 0 THEN
	                    #MissionCode := 0;
	                    #MCRequested := 0;
	                    #Dispatcher["_master"] := 0;
	                    #MissionCode := 0;
	                END_IF;

	                ///////////////////////////
	            200: //MISSION_UnloadPallet_MC1 or MC2
	                // TRE RAMI (17/9): a flangia nuda Gripper_ID[1]=0 e' diverso da
	                // qualunque pinza richiesta, quindi partiva lo scarico di una
	                // pinza inesistente -> query con id=0 -> 990. Vedi nota al 100.
	                IF #Gripper_ID[1] <> #GripperRequested AND #Gripper_ID[1] > 0 THEN
	                    #Dispatcher["_Gripper_Robot_to_TRAY"] := 10;
	                    #Dispatcher["_master"] := 210;
	                ELSIF #Gripper_ID[1] = 0 THEN
	                    #Dispatcher["_Gripper_TRAY_to_Robot"] := 10;
	                    #Dispatcher["_master"] := 220;
	                ELSE
	                    #Dispatcher["_master"] := 220;
	                END_IF;
	            210:
	                IF #Gripper_ID[1] = 0 AND #Dispatcher["_Gripper_Robot_to_TRAY"] = 0 THEN
	                    #Dispatcher["_Gripper_TRAY_to_Robot"] := 10;
	                    #Dispatcher["_master"] := 220;
	                END_IF;

	            220: //gripper OK -> start mission
	                IF #Gripper_ID[1] = #GripperRequested AND #Dispatcher["_Gripper_TRAY_to_Robot"] = 0 THEN
	                    #Dispatcher["_Pallet_MC_to_Robot"] := 10;
	                    #Dispatcher["_master"] := 230;
	                END_IF;
	            230:
	                IF #GripperOccuped[1] AND "DB_RobotMissionStatus".StatusCode = "cmd_executed" AND #Dispatcher["_Pallet_MC_to_Robot"] = 0 THEN
	                    #Dispatcher["_Pallet_Robot_to_TRAY"] := 10;
	                    "DB_RobotMission".Command := 0;  ///\\\

	                    #Dispatcher["_master"] := 240;
	                END_IF;
	            240: //Mission ended
	                IF #Dispatcher["_Pallet_Robot_to_TRAY"] = 0 THEN
	                    #MissionCode := 0;
	                    #MCRequested := 0;
	                    #Dispatcher["_master"] := 0;
	                    #MissionCode := 0;
	                END_IF;

	                ///////////////////////////
	            300: //MissionLoadPart_MC1 or MC2
	                // TRE RAMI (17/9): vedi nota al 100.
	                IF #Gripper_ID[1] <> #GripperRequested AND #Gripper_ID[1] > 0 THEN
	                    #Dispatcher["_Gripper_Robot_to_TRAY"] := 10;
	                    #Dispatcher["_master"] := 310;
	                ELSIF #Gripper_ID[1] = 0 THEN
	                    #Dispatcher["_Gripper_TRAY_to_Robot"] := 10;
	                    #Dispatcher["_master"] := 320;
	                ELSE
	                    #Dispatcher["_master"] := 320;
	                END_IF;
	            310:
	                IF #Gripper_ID[1] = 0 AND #Dispatcher["_Gripper_Robot_to_TRAY"] = 0 THEN
	                    #Dispatcher["_Gripper_TRAY_to_Robot"] := 10;
	                    #Dispatcher["_master"] := 320;
	                END_IF;

	            320: //gripper OK -> start mission
	                IF #Gripper_ID[1] = #GripperRequested AND
	                    #Dispatcher["_Gripper_TRAY_to_Robot"] = 0 THEN

	                    IF NOT #GripperOccuped[1] THEN
	                        #Dispatcher["_Part_TRAY_to_Robot"] := 10;
	                    END_IF;
	                    #Dispatcher["_master"] := 330;
	                END_IF;
	            330:
	                IF #GripperOccuped[1] AND
	                    "DB_RobotMissionStatus".StatusCode = "cmd_waitingNewCmd" AND
	                    #Dispatcher["_Part_TRAY_to_Robot"] = 0
	                THEN
	                    #Dispatcher["_Part_Robot_to_MC"] := 10;
	                    "DB_RobotMission".Command := 0;  ///\\\

	                    #Dispatcher["_master"] := 340;
	                END_IF;
	            340: //Mission ended
	                IF #Dispatcher["_Part_Robot_to_MC"] = 0 THEN
	                    #MissionCode := 0;
	                    #MCRequested := 0;
	                    #Dispatcher["_master"] := 0;
	                    #MissionCode := 0;
	                END_IF;

	                ///////////////////////////
	            400: //MissionUnloadPart_MC1 or MC2
	                // TRE RAMI (17/9): vedi nota al 100.
	                IF #Gripper_ID[1] <> #GripperRequested AND #Gripper_ID[1] > 0 THEN
	                    #Dispatcher["_Gripper_Robot_to_TRAY"] := 10;
	                    #Dispatcher["_master"] := 410;
	                ELSIF #Gripper_ID[1] = 0 THEN
	                    #Dispatcher["_Gripper_TRAY_to_Robot"] := 10;
	                    #Dispatcher["_master"] := 420;
	                ELSE
	                    #Dispatcher["_master"] := 420;
	                END_IF;
	            410:
	                IF #Gripper_ID[1] = 0 AND
	                    #Dispatcher["_Gripper_Robot_to_TRAY"] = 0
	                THEN
	                    #Dispatcher["_Gripper_TRAY_to_Robot"] := 10;
	                    #Dispatcher["_master"] := 420;
	                END_IF;

	            420: //gripper OK -> start mission
	                IF #Gripper_ID[1] = #GripperRequested AND
	                    #Dispatcher["_Gripper_TRAY_to_Robot"] = 0
	                THEN
	                    #Dispatcher["_Part_MC_to_Robot"] := 10;
	                    #Dispatcher["_master"] := 430;
	                END_IF;

	            430:
	                IF ("DB_RobotMissionStatus".StatusCode = "cmd_executed" OR
	                    "DB_RobotMissionStatus".StatusCode = "cmd_waitingNewCmd") AND
	                    #Dispatcher["_Part_MC_to_Robot"] = 0
	                THEN
	                    IF #GripperOccuped[1] AND #GripperOccuped[2] THEN
	                        // entrambi i lati pieni: la macchina sceglie la prossima mossa
	                        "DB_RobotMission".Command := 0;  ///\\\
	                        #MissionCode := 0;
	                        #MCRequested := 0;

	                        #Dispatcher["_master"] := 0;
	                    ELSIF #GripperOccuped[1] OR #GripperOccuped[2] THEN
	                        // UN SOLO LATO PIENO, quale che sia: si deposita.
	                        // Prima la condizione era "GripperOccuped[1] AND NOT [2]":
	                        // col finito prelevato dal LATO 2 (caso normale del ciclo
	                        // automatico, lato 1 libero perche' il grezzo e' gia' in
	                        // macchina) nessun ramo scattava e la catena restava
	                        // appesa qui (visto 5/9).
	                        #Dispatcher["_Part_Robot_to_TRAY"] := 10;
	                        "DB_RobotMission".Command := 0;  ///\\\

	                        #Dispatcher["_master"] := 440;
	                    END_IF;
	                END_IF;

	            440: //Mission ended
	                IF #Dispatcher["_Part_Robot_to_TRAY"] = 0
	                THEN
	                    #MissionCode := 0;
	                    #MCRequested := 0;
	                    #Dispatcher["_master"] := 0;
	                    #MissionCode := 0;
	                END_IF;

	                ///////////////////////////
	            500: //MISSION_LoadPartOnRobot
	                // TRE RAMI (17/9): vedi nota al 100.
	                IF #Gripper_ID[1] <> #GripperRequested AND #Gripper_ID[1] > 0 THEN
	                    #Dispatcher["_Gripper_Robot_to_TRAY"] := 10;
	                    #Dispatcher["_master"] := 510;
	                ELSIF #Gripper_ID[1] = 0 THEN
	                    #Dispatcher["_Gripper_TRAY_to_Robot"] := 10;
	                    #Dispatcher["_master"] := 520;
	                ELSE
	                    #Dispatcher["_master"] := 520;
	                END_IF;
	            510:
	                IF #Gripper_ID[1] = 0 AND
	                    #Dispatcher["_Gripper_Robot_to_TRAY"] = 0
	                THEN
	                    #Dispatcher["_Gripper_TRAY_to_Robot"] := 10;
	                    #Dispatcher["_master"] := 520;
	                END_IF;

	            520: //gripper OK -> start mission
	                IF #Gripper_ID[1] = #GripperRequested AND #Dispatcher["_Gripper_TRAY_to_Robot"] = 0 THEN
	                    #Dispatcher["_Part_TRAY_to_Robot"] := 10;
	                    #Dispatcher["_master"] := 530;
	                END_IF;
	            530:
	                IF #Dispatcher["_Part_TRAY_to_Robot"] = 100 THEN                 //MISSION SUSPENDED FOR WAIT TRAY
	                    IF "DB_BOX_1".ExtractedTray <> "DB_BOX_1".RequestedTray AND
	                        #MissionCode = "MISSION_ExtractTray" AND
	                        #Dispatcher["Extract_TRAY"] = 0
	                    THEN
	                        //HERE ONLY IF WAREHOUSE IS A EASYBOX
	                        //start extract tray
	                        #Dispatcher["Extract_TRAY"] := 10;
	                    END_IF;
	                ELSE
	                    IF #GripperOccuped[1] AND
	                        ("DB_RobotMissionStatus".StatusCode = "cmd_executed" OR
	                        "DB_RobotMissionStatus".StatusCode = "cmd_waitingNewCmd") AND
	                        #Dispatcher["_Part_TRAY_to_Robot"] = 0 THEN
	                        "DB_RobotMission".Command := 0;  ///\\\
	                        #MissionCode := 0;
	                        #MCRequested := 0;
	                        #Dispatcher["_master"] := 0;
	                        #MissionCode := 0;
	                    END_IF;
	                END_IF;

	                ///////////////////////////
	            600: //MISSION_UnloadPartOnRobot
	                // SI SCARICA CON LA PINZA CHE C'E' (5/10). Il confronto con
	                // GripperRequested era un residuo: FB204 lancia questa missione da 35,
	                // 52, 58, 95 e 104 senza impostarlo, dopo un riavvio vale 0 e il ramo
	                // gancio di get_TCP_Data lo azzera. Il master restava qui per sempre,
	                // senza errore. Part_Robot_to_TRAY non lo usa: lo si allinea alla pinza
	                // a bordo e si parte.
	                IF #Gripper_ID[1] > 0 THEN
	                    #GripperRequested := #Gripper_ID[1];
	                    #Dispatcher["_Part_Robot_to_TRAY"] := 10;
	                    #Dispatcher["_master"] := 630;
	                ELSE
	                    #Error := 964;   // scarico pezzo senza pinza registrata a bordo
	                    #MissionCode := 0;
	                    #Dispatcher["_master"] := 0;
	                END_IF;
	            630:
	                // LATO CONFRONTATO, NON USATO COME INDICE (5/10). Gripper_Side vale 0
	                // dopo STOP->RUN (DB_RobotMission non ritentivo) finche' il 30 di
	                // Part_Robot_to_TRAY non lo scrive, e questo stato lo legge prima:
	                // GripperOccuped[0] e' fuori dall'array [1..2], errore di accesso.
	                // Prima il 600 restava fermo dopo un riavvio e qui non si arrivava.
	                IF (("DB_RobotMission".Gripper_Side = 1 AND NOT #GripperOccuped[1])
	                    OR ("DB_RobotMission".Gripper_Side = 2 AND NOT #GripperOccuped[2]))
	                    AND ("DB_RobotMissionStatus".StatusCode = "cmd_executed" OR "DB_RobotMissionStatus".StatusCode = "cmd_waitingNewCmd")
	                    AND #Dispatcher["_Part_Robot_to_TRAY"] = 0
	                THEN
	                    "DB_RobotMission".Command := 0;  ///\\\
	                    #MissionCode := 0;
	                    #MCRequested := 0;
	                    #Dispatcher["_master"] := 0;
	                ELSIF #Dispatcher["_Part_Robot_to_TRAY"] = 0
	                    AND (#Error <> 0
	                    OR ("DB_RobotMission".Gripper_Side <> 1 AND "DB_RobotMission".Gripper_Side <> 2))
	                THEN
	                    // la catena ha chiuso in errore (es. 949 porta operatore aperta)
	                    // prima di scrivere il lato: si chiude la missione, resta l'errore
	                    "DB_RobotMission".Command := 0;
	                    #MissionCode := 0;
	                    #MCRequested := 0;
	                    #Dispatcher["_master"] := 0;
	                END_IF;

	                ///////////////////////////
	            700: //MISSION_ExtractTray
	                IF #Gripper_ID[1] = 0 AND #Gripper_ID[2] = 0 THEN
	                    #Dispatcher["_Gripper_Hook_Search"] := 10;

	                    #Dispatcher["_master"] := 710;
	                ELSE
	                    #Dispatcher["_master"] := 730;
	                END_IF;
	            710: //gripper hook found
	                IF #Dispatcher["_Gripper_Hook_Search"] = 0 THEN
	                    #Dispatcher["_Gripper_TRAY_to_Robot"] := 10;

	                    #Dispatcher["_master"] := 720;
	                END_IF;
	            720: //gripper loaded
	                IF #Dispatcher["_Gripper_TRAY_to_Robot"] = 0 THEN
	                    #Dispatcher["_master"] := 730;
	                END_IF;
	            730: //start extract tray
	                #Dispatcher["Extract_TRAY"] := 10;
	                #Dispatcher["_master"] := 750;

	            750:// extract tray finished
	                // CHIUDE ANCHE IN ERRORE (19/9): la condizione era
	                // "Extract_TRAY = 0 AND #Error = 0". Se un errore si alzava
	                // durante l'estrazione, la catena chiudeva ma questo stato
	                // smetteva di guardarla e MissionCode restava a 200 per sempre.
	                // Da li' la sincronizzazione di FB8 — che pretende MissionCode = 0 —
	                // non girava piu', ExtractedTray restava disallineato dai sensori,
	                // il check posizione rigenerava l'errore a ogni scan e il 949
	                // tornava subito dopo ogni reset. Visto in campo.
	                IF #Dispatcher["Extract_TRAY"] = 0 THEN
	                    #MissionCode := 0;

	                    #Dispatcher["_master"] := 0;
	                END_IF;

	                ///////////////////////////
	            800://MISSION_ReleaseTray
	                IF #Dispatcher["Release_TRAY"] > 10 THEN
	                    #Dispatcher["_master"] := 810;
	                ELSIF #Dispatcher["Release_TRAY"] = 0 THEN
	                    // CHIUSURA SE IL 10 HA GIA' RIFIUTATO (5/10): porta aperta (949),
	                    // pinza assente (2022) o nessun cassetto fuori (20001) portano la
	                    // catena a 0 nello stesso scan in cui la si lancia. L'800 aspettava
	                    // "> 10" per sempre e MissionCode restava a 203.
	                    #MissionCode := 0;
	                    #Dispatcher["_master"] := 0;
	                END_IF;
	            810:
	                // CHIUDE ANCHE IN ERRORE (19/9): vedi nota al 750.
	                IF #Dispatcher["Release_TRAY"] = 0 THEN
	                    #MissionCode := 0;

	                    #Dispatcher["_master"] := 0;
	                END_IF;
	                ///////////////////////////
	            900://"MISSION_UnloadGripper"
	                IF #Dispatcher["_Gripper_Robot_to_TRAY"] = 0 AND #Error = 0 THEN
	                    #MissionCode := 0;

	                    #Dispatcher["_master"] := 0;
	                END_IF;
	                ///////////////////////////
	            950://"MISSION_LoadGripper"
	                IF #Dispatcher["_Gripper_TRAY_to_Robot"] = 0 AND #Error = 0 THEN
	                    #Dispatcher["get_TCP_Data"] := 10;
	                    #Dispatcher["_master"] := 960;
	                END_IF;

	            960: //WAIT end update data
	                IF #Dispatcher["get_TCP_Data"] = 0 THEN
	                    #MissionCode := 0;

	                    #Dispatcher["Reset_or_log_MissionData"] := 10;
	                    #Dispatcher["_master"] := 0;

	                END_IF;

	                //////////////////////
	            970: // SWAP fase A: query slot di casa della pinza a bordo
	                IF "SqlCommands".sqlCommands[0] = '' THEN
	                    #queryTemp := CONCAT(IN1 := 'SELECT X,Y,Z,X_ROT,Y_ROT,Z_ROT,APPROACH_TYPE,APPROACH_X,APPROACH_Y,APPROACH_Z from COORDINATES_GRIPPER_SHELF where id=',
	                                         IN2 := "INT_TO_STRING_WITHOUT_SIGN"(#Gripper_ID[1]));
	                    #queryStartExecution := TRUE;
	                    #Dispatcher["_master"] := 971;
	                END_IF;
	            971: // presa in carico query VERIFICATA
	                // SqlData e' un buffer unico condiviso: senza il confronto su
	                // sqlCommands[0] il 972 puo' leggere la risposta di un altro
	                // richiedente e mandare il robot su coordinate altrui.
	                IF NOT "DB_executeQuery".readyForNextQuery
	                    AND "SqlCommands".sqlCommands[0] = #queryTemp THEN
	                    #Dispatcher["_master"] := 972;
	                END_IF;
	            972: // frame A (deposito) + comando 17
	                IF "DB_executeQuery".dataReady AND "DB_executeQuery".noData THEN
	                    // slot di casa della pinza a bordo non trovato: con FB6 corretto
	                    // "zero righe" non e' piu' dataError, va intercettato qui.
	                    #Error := 990;
	                    "DB_executeQuery".readyForNextQuery := TRUE;
	                    #MissionCode := 0;
	                    #Dispatcher["_master"] := 0;
	                ELSIF "DB_executeQuery".dataReady AND NOT "DB_executeQuery".dataError THEN
	                    "DB_RobotMission"."X_Pick-Place" := "SqlData".data.rows[0].col[0];
	                    "DB_RobotMission"."Y_Pick-Place" := "SqlData".data.rows[0].col[1];
	                    "DB_RobotMission"."Z_Pick-Place" := "SqlData".data.rows[0].col[2];
	                    "DB_RobotMission"."XRot_Pick-Place" := "SqlData".data.rows[0].col[3];
	                    "DB_RobotMission"."YRot_Pick-Place" := "SqlData".data.rows[0].col[4];
	                    "DB_RobotMission"."ZRot_Pick-Place" := "SqlData".data.rows[0].col[5];
	                    "DB_RobotMission".X_approach := "SqlData".data.rows[0].col[7];
	                    "DB_RobotMission".Y_approach := "SqlData".data.rows[0].col[8];
	                    "DB_RobotMission".Z_approach := "SqlData".data.rows[0].col[9];
	                    "DB_RobotMission".XRot_approach := 0;
	                    "DB_RobotMission".YRot_approach := 0;
	                    "DB_RobotMission".ZRot_approach := 0;
	                    "DB_RobotMission".ApproachType := "FC_ExtractApproach"(approachVal := "SqlData".data.rows[0].col[6], pick := FALSE);
	                    "DB_RobotMission".Object_Type := "Gripper";
	                    "DB_RobotMission".Unit_code := "Warehouse1";
	                    "DB_RobotMission".Gripper_Side := 1;
	                    "DB_RobotMission".Gripper_code := #Gripper_ID[1];
	                    "DB_executeQuery".readyForNextQuery := TRUE;

	                    "DB_RobotMission".Command := "CMD_RobotSwapGripper";
	                    #Dispatcher["_master"] := 973;
	                ELSIF "DB_executeQuery".dataError THEN
	                    #Error := 990;
	                    "DB_executeQuery".readyForNextQuery := TRUE;
	                    #MissionCode := 0;
	                    #Dispatcher["_master"] := 0;
	                END_IF;
	            973: // attesa acquisizione robot
	                IF "DB_RobotMissionStatus".StatusCode = "cmd_acquired" OR
	                    "DB_RobotMissionStatus".StatusCode = "cmd_executing" THEN
	                    #Dispatcher["_master"] := 974;
	                END_IF;
	            974: // deposito eseguito: il robot alza REQ_FASE2 restando in executing
	                IF "Robot_SwapPhase2Req" AND NOT "Gripper_mounted" THEN
	                    #Gripper_ID[1] := 0;                       // registro di meta' corsa: la vecchia e' a terra
	                    #Gripper_ID[2] := 0;
	                    #Dispatcher["updateGripperOnRobot"] := 10; // DB e pannello sanno subito
	                    #Dispatcher["_master"] := 975;
	                END_IF;
	            975: // query slot della pinza nuova
	                IF #Dispatcher["updateGripperOnRobot"] = 0 AND "SqlCommands".sqlCommands[0] = '' THEN
	                    #queryTemp := CONCAT(IN1 := 'SELECT X,Y,Z,X_ROT,Y_ROT,Z_ROT,APPROACH_TYPE,APPROACH_X,APPROACH_Y,APPROACH_Z from COORDINATES_GRIPPER_SHELF where id=',
	                                         IN2 := "INT_TO_STRING_WITHOUT_SIGN"(#GripperRequested));
	                    #queryStartExecution := TRUE;
	                    #Dispatcher["_master"] := 976;
	                END_IF;
	            976: // presa in carico query VERIFICATA
	                // SqlData e' un buffer unico condiviso: senza il confronto su
	                // sqlCommands[0] il 977 puo' leggere la risposta di un altro
	                // richiedente. Qui e' particolarmente critico: la pinza vecchia
	                // e' gia' a terra e il robot sta per andare a prendere la nuova.
	                IF NOT "DB_executeQuery".readyForNextQuery
	                    AND "SqlCommands".sqlCommands[0] = #queryTemp THEN
	                    #Dispatcher["_master"] := 977;
	                END_IF;
	            977: // frame B (prelievo) + DATI_PRONTI
	                IF "DB_executeQuery".dataReady AND "DB_executeQuery".noData THEN
	                    // slot della pinza nuova non trovato: con FB6 corretto "zero
	                    // righe" non e' piu' dataError, va intercettato qui.
	                    // NB: pinza vecchia gia' a terra e registrata: stato coerente.
	                    #Error := 990;
	                    "DB_executeQuery".readyForNextQuery := TRUE;
	                    #MissionCode := 0;
	                    #Dispatcher["_master"] := 0;
	                ELSIF "DB_executeQuery".dataReady AND NOT "DB_executeQuery".dataError THEN
	                    "DB_RobotMission"."X_Pick-Place" := "SqlData".data.rows[0].col[0];
	                    "DB_RobotMission"."Y_Pick-Place" := "SqlData".data.rows[0].col[1];
	                    "DB_RobotMission"."Z_Pick-Place" := "SqlData".data.rows[0].col[2];
	                    "DB_RobotMission"."XRot_Pick-Place" := "SqlData".data.rows[0].col[3];
	                    "DB_RobotMission"."YRot_Pick-Place" := "SqlData".data.rows[0].col[4];
	                    "DB_RobotMission"."ZRot_Pick-Place" := "SqlData".data.rows[0].col[5];
	                    "DB_RobotMission".X_approach := "SqlData".data.rows[0].col[7];
	                    "DB_RobotMission".Y_approach := "SqlData".data.rows[0].col[8];
	                    "DB_RobotMission".Z_approach := "SqlData".data.rows[0].col[9];
	                    "DB_RobotMission".XRot_approach := 0;
	                    "DB_RobotMission".YRot_approach := 0;
	                    "DB_RobotMission".ZRot_approach := 0;
	                    "DB_RobotMission".ApproachType := "FC_ExtractApproach"(approachVal := "SqlData".data.rows[0].col[6], pick := TRUE);
	                    "DB_RobotMission".Object_Type := "Gripper";
	                    "DB_RobotMission".Unit_code := "Warehouse1";
	                    "DB_RobotMission".Gripper_Side := 1;
	                    "DB_RobotMission".Gripper_code := #GripperRequested;
	                    "DB_executeQuery".readyForNextQuery := TRUE;

	                    #swapDataReady := TRUE;          // -> Option_free verso il robot
	                    #Dispatcher["_master"] := 978;
	                ELSIF "DB_executeQuery".dataError THEN
	                    #Error := 990;
	                    "DB_executeQuery".readyForNextQuery := TRUE;
	                    // NB: pinza vecchia gia' a terra e registrata: stato coerente, missione morta qui
	                    #MissionCode := 0;
	                    #Dispatcher["_master"] := 0;
	                END_IF;
	            978: // esito prelievo: doppia conferma (esito + sensore)
	                IF "DB_RobotMissionStatus".StatusCode = "cmd_executed" AND "Gripper_mounted" THEN
	                    #swapDataReady := FALSE;
	                    "DB_RobotMission".Command := 0;
	                    // REGISTRI E DATABASE LI SCRIVE LA CATENA UNICA (17/9): e' lei
	                    // che cerca la gemella. Prima il 978 scriveva solo il lato 1 e
	                    // il lato 2 restava a zero — e siccome il 35 di FB204 cambia
	                    // pinza SEMPRE via swap, in ciclo automatico la pinza doppia
	                    // veniva usata come singola: niente missione 16, finito preso
	                    // col lato 1, e l'operatore costretto a dichiararlo a mano.
	                    #Dispatcher["_Set_Gripper_OnBoard"] := 10;
	                    #Dispatcher["_master"] := 9781;
	                END_IF;

	            9781: // attesa registrazione conclusa
	                IF #Dispatcher["_Set_Gripper_OnBoard"] = 0 THEN
	                    #Dispatcher["_master"] := 979;
	                END_IF;

	            979: // update chiuso + robot libero -> aggiornamento TCP
	                // La guardia su updateGripperOnRobot e' ridondante — la catena
	                // _Set_Gripper_OnBoard al 50 aspetta gia' che l'update chiuda —
	                // ma costa niente e rende lo stato leggibile da solo: qui si
	                // prosegue solo con database allineato E robot libero.
	                IF #Dispatcher["updateGripperOnRobot"] = 0 AND
	                    "DB_RobotMissionStatus".StatusCode = "cmd_waitingNewCmd" THEN
	                    #Dispatcher["get_TCP_Data"] := 10;
	                    #Dispatcher["_master"] := 980;
	                END_IF;
	            980: // TCP chiuso -> fine missione
	                IF #Dispatcher["get_TCP_Data"] = 0 THEN
	                    #Dispatcher["Reset_or_log_MissionData"] := 10;
	                    #Dispatcher["_master"] := 985;
	                END_IF;
	            985: // ri-assert del codice pinza dopo il reset (il registro è la verità)
	                IF #Dispatcher["Reset_or_log_MissionData"] = 0 THEN
	                    "DB_RobotMission".Gripper_code := #Gripper_ID[1];
	                    #MissionCode := 0;
	                    #Dispatcher["_master"] := 0;
	                END_IF;

	                //////////////////////
	            1000: //MISSION_Load_Pallet
	                #Dispatcher["_Gripper4Pallet_Search"] := 10;
	                #Dispatcher["_master"] := 1010;

	            1010:
	                IF #Dispatcher["_Gripper4Pallet_Search"] = 0 THEN
	                    IF #GripperRequested > 0 THEN
	                        IF #GripperRequested <> #Gripper_ID[1] AND #Gripper_ID[1] > 0 THEN
	                            #Dispatcher["_Gripper_Robot_to_TRAY"] := 10;
	                            #Dispatcher["_master"] := 1020;
	                        ELSE
	                            #Dispatcher["_master"] := 1050;
	                        END_IF;
	                    ELSE
	                        #Error := "_Gripper4Pallet_Search" * 100 + 22;
	                    END_IF;
	                END_IF;

	            1020:
	                IF #Dispatcher["_Gripper_Robot_to_TRAY"] = 0 THEN
	                    #Dispatcher["_Gripper_TRAY_to_Robot"] := 10;
	                    #Dispatcher["_master"] := 1050;
	                END_IF;
	            1050:
	                IF #Dispatcher["_Gripper_TRAY_to_Robot"] = 0 THEN
	                    #Dispatcher["_Pallet_TRAY_to_Robot"] := 10;
	                    #Dispatcher["_master"] := 1060;
	                END_IF;
	            1060:
	                IF #Dispatcher["_Pallet_TRAY_to_Robot"] = 0 THEN
	                    #MissionCode := 0;
	                    #Dispatcher["_master"] := 0;
	                END_IF;
	                //////////////////////
	            1500: //MISSION_Unload_Pallet  (HMI command)
	                IF #Gripper_ID[1] = 0 THEN
	                    #Error := "MISSION_Unload_Pallet" * 100 + 22;
	                ELSIF NOT #GripperOccuped[1] THEN
	                    #Error := "MISSION_Unload_Pallet" * 100 + 23;
	                ELSE
	                    #Dispatcher["_master"] := 1510;
	                END_IF;

	                ///////////// 1100: pick pezzo da cassetto (HMI)
	            1100: // swap pinza se serve (pattern catene auto)
	                IF #Gripper_ID[1] <> #GripperRequested AND #Gripper_ID[1] > 0 THEN
	                    #Dispatcher["_Gripper_Robot_to_TRAY"] := 10;
	                    #Dispatcher["_master"] := 1110;
	                ELSIF #Gripper_ID[1] = 0 THEN
	                    #Dispatcher["_Gripper_TRAY_to_Robot"] := 10;
	                    #Dispatcher["_master"] := 1115;
	                ELSE
	                    #Dispatcher["_master"] := 1120;
	                END_IF;
	            1110: // scarico pinza attuale
	                IF #Gripper_ID[1] = 0 AND #Dispatcher["_Gripper_Robot_to_TRAY"] = 0 THEN
	                    #Dispatcher["_Gripper_TRAY_to_Robot"] := 10;
	                    #Dispatcher["_master"] := 1115;
	                END_IF;
	            1115: // carico pinza richiesta
	                IF #Dispatcher["_Gripper_TRAY_to_Robot"] = 0 THEN
	                    #Dispatcher["_master"] := 1120;
	                END_IF;
	            1120: // pinza ok -> preleva pezzo
	                IF #Gripper_ID[1] = #GripperRequested THEN
	                    #Dispatcher["_Part_TRAY_to_Robot"] := 10;
	                    #Dispatcher["_master"] := 1130;
	                END_IF;
	            1130: // fine
	                IF #Dispatcher["_Part_TRAY_to_Robot"] = 0 AND #Error = 0 THEN
	                    #MissionCode := 0;
	                    #MCRequested := 0;
	                    #Dispatcher["_master"] := 0;
	                END_IF;

	                ///////////// 1150: place pezzo in cassetto (HMI)
	            1150:
	                IF #Dispatcher["_Part_Robot_to_TRAY"] = 0 AND #Error = 0 THEN
	                    #MissionCode := 0;
	                    #MCRequested := 0;
	                    #Dispatcher["_master"] := 0;
	                END_IF;

	                ///////////// 1200: pick pezzo da MC1 (HMI)
	            1200: // swap pinza se serve
	                IF #Gripper_ID[1] <> #GripperRequested AND #Gripper_ID[1] > 0 THEN
	                    #Dispatcher["_Gripper_Robot_to_TRAY"] := 10;
	                    #Dispatcher["_master"] := 1210;
	                ELSIF #Gripper_ID[1] = 0 THEN
	                    #Dispatcher["_Gripper_TRAY_to_Robot"] := 10;
	                    #Dispatcher["_master"] := 1215;
	                ELSE
	                    #Dispatcher["_master"] := 1220;
	                END_IF;
	            1210:
	                IF #Gripper_ID[1] = 0 AND #Dispatcher["_Gripper_Robot_to_TRAY"] = 0 THEN
	                    #Dispatcher["_Gripper_TRAY_to_Robot"] := 10;
	                    #Dispatcher["_master"] := 1215;
	                END_IF;
	            1215:
	                IF #Dispatcher["_Gripper_TRAY_to_Robot"] = 0 THEN
	                    #Dispatcher["_master"] := 1220;
	                END_IF;
	            1220:
	                IF #Gripper_ID[1] = #GripperRequested THEN
	                    #Dispatcher["_Part_MC_to_Robot"] := 10;
	                    #Dispatcher["_master"] := 1230;
	                END_IF;
	            1230:
	                IF #Dispatcher["_Part_MC_to_Robot"] = 0 AND #Error = 0 THEN
	                    #MissionCode := 0;
	                    #MCRequested := 0;
	                    #Dispatcher["_master"] := 0;
	                END_IF;

	                ///////////// 1250: place pezzo su MC1 (HMI)
	            1250:
	                IF #Dispatcher["_Part_Robot_to_MC"] = 0 AND #Error = 0 THEN
	                    #MissionCode := 0;
	                    #MCRequested := 0;
	                    #Dispatcher["_master"] := 0;
	                END_IF;

	                ///////////// 1300: pick pallet da MC1 (HMI)
	            1300: // pinza giusta dal pallet (come 1000 warehouse)
	                #Dispatcher["_Gripper4Pallet_Search"] := 10;
	                #Dispatcher["_master"] := 1310;
	            1310:
	                IF #Dispatcher["_Gripper4Pallet_Search"] = 0 THEN
	                    IF #GripperRequested > 0 THEN
	                        IF #GripperRequested <> #Gripper_ID[1] AND #Gripper_ID[1] > 0 THEN
	                            #Dispatcher["_Gripper_Robot_to_TRAY"] := 10;
	                            #Dispatcher["_master"] := 1320;
	                        ELSIF #Gripper_ID[1] = 0 THEN
	                            #Dispatcher["_Gripper_TRAY_to_Robot"] := 10;
	                            #Dispatcher["_master"] := 1330;
	                        ELSE
	                            #Dispatcher["_master"] := 1340;
	                        END_IF;
	                    ELSE
	                        #Error := "_Gripper4Pallet_Search" * 100 + 22;
	                    END_IF;
	                END_IF;
	            1320:
	                IF #Dispatcher["_Gripper_Robot_to_TRAY"] = 0 THEN
	                    #Dispatcher["_Gripper_TRAY_to_Robot"] := 10;
	                    #Dispatcher["_master"] := 1330;
	                END_IF;
	            1330:
	                IF #Dispatcher["_Gripper_TRAY_to_Robot"] = 0 THEN
	                    #Dispatcher["_master"] := 1340;
	                END_IF;
	            1340:
	                IF #Gripper_ID[1] = #GripperRequested THEN
	                    #Dispatcher["_Pallet_MC_to_Robot"] := 10;
	                    #Dispatcher["_master"] := 1345;
	                END_IF;
	            1345:
	                IF #Dispatcher["_Pallet_MC_to_Robot"] = 0 AND #Error = 0 THEN
	                    #MissionCode := 0;
	                    #MCRequested := 0;
	                    #Dispatcher["_master"] := 0;
	                END_IF;

	                ///////////// 1350: place pallet su MC1 (HMI)
	            1350:
	                IF #Dispatcher["_Pallet_Robot_to_MC"] = 0 AND #Error = 0 THEN
	                    #MissionCode := 0;
	                    #MCRequested := 0;
	                    #Dispatcher["_master"] := 0;
	                END_IF;
	                ///////////// 1400: prelievo finito + deposito grezzo in MC (comando robot 16)
	                // Un solo ingresso in macchina: il robot arriva col grezzo sul lato 1,
	                // preleva il finito col lato 2, ruota, deposita il grezzo.
	                // Handshake a due fasi come lo swap pinza: il robot alza
	                // Robot_SwapPhase2Req, il PLC manda il frame di deposito e Ok_Phase2_MC.
	            1400: // query unica: entrambe le quote dalla stessa posizione MC.
	                // Il calcolo sta nella vista COORDINATES_PICKPLACE_MC: la query
	                // composta a mano superava i 254 caratteri di queryTemp e arrivava
	                // TRONCATA a SQL -> zero righe -> 13599 (visto 15/9). Il 1401 non
	                // se ne accorge perche' confronta con la stessa stringa tagliata.
	                // Z_PICK_MC = prelievo del FINITO (Z_PLACE del pezzo)
	                // Z_PLACE_MC = deposito del GREZZO (Z_PICK del pezzo)
	                IF "SqlCommands".sqlCommands[0] = '' THEN
	                    IF NOT #GripperOccuped[1] THEN
	                        #Error := "MISSION_PickPlacePart_MC" * 100 + 23;   // nessun grezzo a bordo
	                        #MissionCode := 0;
	                        #Dispatcher["_master"] := 0;
	                    ELSIF #GripperOccuped[2] THEN
	                        #Error := "MISSION_PickPlacePart_MC" * 100 + 21;   // lato finito gia' occupato
	                        #MissionCode := 0;
	                        #Dispatcher["_master"] := 0;
	                    ELSIF "DB_MC1".io_in.viceOpened THEN
	                        // MORSA APERTA = NESSUN FINITO DA PRELEVARE (17/9).
	                        // Stessa guardia del 10 di Part_MC_to_Robot: la 16 entra in
	                        // macchina per prelevare E depositare, senza pezzo da
	                        // prendere la sequenza a due fasi non ha senso.
	                        #Error := 894;
	                        #MissionCode := 0;
	                        #Dispatcher["_master"] := 0;
	                    ELSIF "DB_MC1".order.ID > 0 THEN
	                        #queryTemp := CONCAT(IN1 := 'select X,Y,Z_PICK_MC,Z_PLACE_MC,X_ROT,Y_ROT,Z_ROT,APPROACH_TYPE,APPROACH_X,APPROACH_Y,APPROACH_Z from COORDINATES_PICKPLACE_MC where ORDER_ID=',
	                                             IN2 := "INT_TO_STRING_WITHOUT_SIGN"(DINT_TO_INT("DB_MC1".order.ID)));
	                        #queryStartExecution := TRUE;
	                        #Dispatcher["_master"] := 1401;
	                    ELSE
	                        // MANUALE: nessun ordine attivo, uso il piu' recente
	                        #queryTemp := 'select top 1 X,Y,Z_PICK_MC,Z_PLACE_MC,X_ROT,Y_ROT,Z_ROT,APPROACH_TYPE,APPROACH_X,APPROACH_Y,APPROACH_Z from COORDINATES_PICKPLACE_MC order by ORDER_ID desc';
	                        #queryStartExecution := TRUE;
	                        #Dispatcher["_master"] := 1401;
	                    END_IF;
	                END_IF;
	            1401: // presa in carico query VERIFICATA
	                // SqlData e' un buffer unico condiviso: senza il confronto su
	                // sqlCommands[0] il 1402 puo' leggere la risposta di un altro
	                // richiedente e mandare al robot quote sbagliate per il prelievo
	                // del finito E per il deposito del grezzo (zPlaceTemp).
	                IF NOT "DB_executeQuery".readyForNextQuery
	                    AND "SqlCommands".sqlCommands[0] = #queryTemp THEN
	                    #Dispatcher["_master"] := 1402;
	                END_IF;
	            1402: // FRAME A: prelievo del finito, lato 2. La missione NON parte qui:
	                // prima si leggono e si congelano le quote di spinta (1410-1414),
	                // perche' il robot non deve aspettare il ponte SQL a pezzo posato.
	                IF "DB_executeQuery".dataReady AND "DB_executeQuery".noData THEN
	                    // quote non trovate (ordine/pezzo/attrezzatura incoerenti a DB):
	                    // con FB6 corretto "zero righe" non e' piu' dataError.
	                    #Error := "MISSION_PickPlacePart_MC" * 100 + 99;
	                    "DB_executeQuery".readyForNextQuery := TRUE;
	                    #MissionCode := 0;
	                    #Dispatcher["_master"] := 0;
	                ELSIF "DB_executeQuery".dataReady AND NOT "DB_executeQuery".dataError THEN
	                    // QUOTE DI DEPOSITO CONGELATE, come zPlaceTemp: il frame B le
	                    // riprende tali e quali. Cosi' la fase di deposito e' identica
	                    // a quella collaudata in Part_Robot_to_MC.
	                    #xPlaceTemp := "SqlData".data.rows[0].col[0];
	                    #zPlaceTemp := "SqlData".data.rows[0].col[3];

	                    // X DI PRELIEVO = quota nominale + CORSA DELLA SPINTA DEL PEZZO
	                    // PRECEDENTE: il finito in macchina puo' esserci stato messo
	                    // con la spinta, e allora non sta dove il deposito lo aveva
	                    // posato. Vale zero se la spinta non c'e' stata.
	                    "DB_RobotMission"."X_Pick-Place" := #xPlaceTemp + #xPushOffsetMC;
	                    "DB_RobotMission"."Y_Pick-Place" := "SqlData".data.rows[0].col[1];
	                    "DB_RobotMission"."Z_Pick-Place" := "SqlData".data.rows[0].col[2];   // Z_PICK
	                    "DB_RobotMission"."XRot_Pick-Place" := "SqlData".data.rows[0].col[4];
	                    "DB_RobotMission"."YRot_Pick-Place" := "SqlData".data.rows[0].col[5];
	                    "DB_RobotMission"."ZRot_Pick-Place" := "SqlData".data.rows[0].col[6];
	                    "DB_RobotMission".X_approach := "SqlData".data.rows[0].col[8];
	                    "DB_RobotMission".Y_approach := "SqlData".data.rows[0].col[9];
	                    "DB_RobotMission".Z_approach := "SqlData".data.rows[0].col[10];
	                    "DB_RobotMission".XRot_approach := 0;
	                    "DB_RobotMission".YRot_approach := 0;
	                    "DB_RobotMission".ZRot_approach := 0;
	                    "DB_RobotMission".ApproachType := "FC_ExtractApproach"(approachVal := "SqlData".data.rows[0].col[7], pick := TRUE);
	                    "DB_RobotMission".Object_Type := "Part";
	                    "DB_RobotMission".Unit_code := #MCRequested + 10;
	                    "DB_RobotMission".Gripper_code := #GripperRequested;
	                    "DB_RobotMission".Gripper_Side := 2;                  // finito
	                    "DB_executeQuery".readyForNextQuery := TRUE;

	                    #xPushTemp := 0;
	                    #xStopTemp := 0;
	                    #Dispatcher["_master"] := 1410;
	                ELSIF "DB_executeQuery".dataError THEN
	                    #Error := "MISSION_PickPlacePart_MC" * 100 + 99;
	                    "DB_executeQuery".readyForNextQuery := TRUE;
	                    #MissionCode := 0;
	                    #Dispatcher["_master"] := 0;
	                END_IF;

	            1403: // attesa acquisizione robot
	                IF "DB_RobotMissionStatus".StatusCode = "cmd_acquired" OR
	                    "DB_RobotMissionStatus".StatusCode = "cmd_executing" THEN
	                    #Dispatcher["_master"] := 1404;
	                END_IF;

	            1404: // il robot ha il finito e chiede la fase 2 -> FRAME B: deposito grezzo, lato 1
	                IF "Robot_Phase2Req_MC" THEN
	                    "DB_RobotMission"."X_Pick-Place" := #xPlaceTemp;      // quota nominale
	                    "DB_RobotMission"."Z_Pick-Place" := #zPlaceTemp;      // Z_PLACE
	                    "DB_RobotMission".Gripper_Side := 1;                  // grezzo
	                    "Ok_Phase2_MC" := TRUE;
	                    IF "Q_PushEnable_MC" THEN
	                        #Dispatcher["_master"] := 1420;
	                    ELSE
	                        #Dispatcher["_master"] := 1405;
	                    END_IF;
	                END_IF;

	            1405: // missione conclusa: aggiorna i registri di bordo
	                IF "DB_RobotMissionStatus".StatusCode = "cmd_executed" THEN
	                    "Ok_Phase2_MC" := FALSE;
	                    "DB_RobotMission".Command := 0;
	                    #GripperOccuped[2] := TRUE;                           // finito a bordo
	                    #GripperOccuped[1] := FALSE;                          // grezzo lasciato in macchina

	                    // CORSA DELLA SPINTA applicata al grezzo appena depositato: il
	                    // prelievo del prossimo giro dovra' andare a prenderlo li'.
	                    IF "Q_PushEnable_MC" THEN
	                        #xPushOffsetMC := #xStopTemp - #xPushTemp;
	                    ELSE
	                        #xPushOffsetMC := 0;
	                    END_IF;

	                    "Q_PushEnable_MC" := FALSE;
	                    "Ok_PushSpinta_MC" := FALSE;
	                    "Ok_PushArrivo_MC" := FALSE;

	                    #Dispatcher["updatePartOnRobot"] := 20 + DINT_TO_INT("FINISHED");
	                    #Dispatcher["_master"] := 1406;
	                END_IF;

	            1406:
	                IF #Dispatcher["updatePartOnRobot"] = 0 THEN
	                    "DB_RobotMission".Gripper_Side := 1;
	                    #Dispatcher["updatePartOnRobot"] := 10 + DINT_TO_INT("EMPTY");
	                    #Dispatcher["_master"] := 1407;
	                END_IF;
	            1407:
	                IF #Dispatcher["updatePartOnRobot"] = 0 THEN
	                    #Dispatcher["updatePartOnMC"] := 10 + DINT_TO_INT("RAW");
	                    #Dispatcher["_master"] := 1408;
	                END_IF;
	            1408: // fine missione
	                IF #Dispatcher["updatePartOnMC"] = 0 THEN
	                    #MissionCode := 0;
	                    #MCRequested := 0;
	                    #Dispatcher["_master"] := 0;
	                END_IF;

	            1410: // SPINTA: query sulle quote di spinta e arrivo per il grezzo che
	                // sta per entrare. Stesso schema dello stato 32 di Part_Robot_to_MC.
	                IF #MCRequested <> 1 THEN
	                    #Dispatcher["_master"] := 1414;          // MC2 non esiste: nessuna spinta
	                ELSIF "SqlCommands".sqlCommands[0] = '' THEN
	                    IF "DB_MC1".order.ID > 0 THEN
	                        #queryTemp := CONCAT(IN1 := 'select X_PUSH,X_STOP from COORDINATES_PUSH_MC where MC=1 and ORDER_ID=',
	                                             IN2 := "INT_TO_STRING_WITHOUT_SIGN"(DINT_TO_INT("DB_MC1".order.ID)));
	                    ELSE
	                        #queryTemp := 'select top 1 X_PUSH,X_STOP from COORDINATES_PUSH_MC where MC=1 order by ORDER_ID desc';
	                    END_IF;
	                    #queryStartExecution := TRUE;
	                    #Dispatcher["_master"] := 1411;
	                END_IF;

	            1411: // presa in carico VERIFICATA della query spinta
	                IF NOT "DB_executeQuery".readyForNextQuery
	                    AND "SqlCommands".sqlCommands[0] = #queryTemp THEN
	                    #Dispatcher["_master"] := 1412;
	                END_IF;

	            1412: // esito spinta con CONTROLLO DI PLAUSIBILITA'.
	                // Il ponte SQL NON converte NULL in zero: restituisce valori
	                // casuali (visto 15/9: -1.056.960.259 con PUSH_STATUS DISABLED).
	                // Il riferimento e' la quota di DEPOSITO congelata.
	                IF "DB_executeQuery".dataReady THEN
	                    IF "DB_executeQuery".noData OR "DB_executeQuery".dataError THEN
	                        #xPushTemp := 0;
	                        #xStopTemp := 0;
	                    ELSE
	                        #xPushTemp := "SqlData".data.rows[0].col[0];
	                        #xStopTemp := "SqlData".data.rows[0].col[1];

	                        IF ABS(#xPushTemp - #xPlaceTemp) > 500000
	                            OR ABS(#xStopTemp - #xPlaceTemp) > 500000
	                        THEN
	                            #xPushTemp := 0;
	                            #xStopTemp := 0;
	                        END_IF;
	                    END_IF;
	                    "DB_executeQuery".readyForNextQuery := TRUE;
	                    #queryTemp := '';
	                    #queryStartExecution := FALSE;
	                    #Dispatcher["_master"] := 1416;
	                END_IF;

	            1416: // SOFFIAGGIO: vedi nota estesa al 37 di Part_Robot_to_MC.
	                // Qui la X di deposito e' xPlaceTemp, congelata al 1402: la
	                // missione ne usa due — prelievo finito e deposito grezzo — e
	                // l'appoggio si calcola sempre su quella di DEPOSITO.
	                IF "SqlCommands".sqlCommands[0] = '' THEN
	                    IF "DB_MC1".order.ID > 0 THEN
	                        #queryTemp := CONCAT(IN1 := 'select CLAW_LENGTH,PART_WIDTH,STOP_BEYOND_CLAW from COORDINATES_BLOW_MC where ORDER_ID=',
	                                             IN2 := "INT_TO_STRING_WITHOUT_SIGN"(DINT_TO_INT("DB_MC1".order.ID)));
	                        #queryStartExecution := TRUE;
	                        #Dispatcher["_master"] := 1417;
	                    ELSE
	                        // nessun ordine attivo: niente da leggere, si prosegue.
	                        // ATTENZIONE: qui va 1414, non 1416 — rimandare a se stesso
	                        // lascia il master appeso per sempre, e tonSwapB non copre
	                        // questo stato.
	                        #Dispatcher["_master"] := 1414;
	                    END_IF;
	                END_IF;

	            1417: // presa in carico VERIFICATA
	                IF NOT "DB_executeQuery".readyForNextQuery
	                    AND "SqlCommands".sqlCommands[0] = #queryTemp THEN
	                    #Dispatcher["_master"] := 1418;
	                END_IF;

	            1418: // esito: scrive le tre variabili PROFINET.
	                // APPOGGIO COME MISURA: vedi nota al 39 di Part_MC_to_Robot.
	                // Qui xPlaceTemp non entra piu': era la quota di deposito, e il
	                // robotista la posizione non la vuole.
	                IF "DB_executeQuery".dataReady THEN
	                    IF NOT "DB_executeQuery".noData AND NOT "DB_executeQuery".dataError THEN
	                        "Vice_ClawLength_mm" := DINT_TO_INT("SqlData".data.rows[0].col[0] / 1000);
	                        "Part_Width_mm" := DINT_TO_INT("SqlData".data.rows[0].col[1] / 1000);
	                        "X_Support_mm" := DINT_TO_INT(("SqlData".data.rows[0].col[0] / 2
	                                                                                    + "SqlData".data.rows[0].col[2]) / 1000);
	                    END_IF;
	                    "DB_executeQuery".readyForNextQuery := TRUE;
	                    #queryTemp := '';
	                    #queryStartExecution := FALSE;
	                    #Dispatcher["_master"] := 1414;
	                END_IF;

	            1414: // consenso alla spinta PRIMA del comando, come al 40 di
	                // Part_Robot_to_MC: il robot lo legge quando acquisisce la
	                // missione e sa quante fasi dovra' chiedere.
	                "Q_PushEnable_MC" := (#xPushTemp <> 0) AND (#xStopTemp <> 0);
	                "Ok_PushSpinta_MC" := FALSE;
	                "Ok_PushArrivo_MC" := FALSE;
	                "Ok_Phase2_MC" := FALSE;

	                "DB_RobotMission".Command := "CMD_RobotPickPlaceObject";
	                #Dispatcher["_master"] := 1403;

	            1420: // SPINTA fase 1: il robot ha depositato e chiede la quota di spinta
	                IF "Robot_PushDepositoFatto_MC" THEN
	                    "DB_RobotMission"."X_Pick-Place" := #xPushTemp;
	                    "Ok_PushSpinta_MC" := TRUE;
	                    #Dispatcher["_master"] := 1421;
	                END_IF;

	            1421: // attesa che il robot abbassi il suo bit: ha letto la quota
	                IF NOT "Robot_PushDepositoFatto_MC" THEN
	                    "Ok_PushSpinta_MC" := FALSE;
	                    #Dispatcher["_master"] := 1422;
	                END_IF;

	            1422: // SPINTA fase 2: il robot e' in posizione e chiede la quota di arrivo
	                IF "Robot_PushInPos_MC" THEN
	                    "DB_RobotMission"."X_Pick-Place" := #xStopTemp;
	                    "Ok_PushArrivo_MC" := TRUE;
	                    #Dispatcher["_master"] := 1423;
	                END_IF;

	            1423: // attesa che il robot abbassi il suo bit: ha letto la quota
	                IF NOT "Robot_PushInPos_MC" THEN
	                    "Ok_PushArrivo_MC" := FALSE;
	                    #Dispatcher["_master"] := 1405;
	                END_IF;

	            1510:
	                #Dispatcher["_Pallet_Robot_to_TRAY"] := 10;
	                #Dispatcher["_master"] := 1520;

	            1520:
	                IF #Dispatcher["_Pallet_Robot_to_TRAY"] = 0 THEN
	                    #MissionCode := 0;
	                    #Dispatcher["_master"] := 0;
	                END_IF;

	                ///////////// 1600: apertura chela lato 1 (HMI)
	            1600:
	                "DB_RobotMission".Gripper_Side := 1;
	                "DB_RobotMission".Gripper_code := #Gripper_ID[1];
	                "DB_RobotMission".Command := "CMD_RobotOpenGripper1";
	                #Dispatcher["_master"] := 1601;
	            1601:
	                IF "DB_RobotMissionStatus".StatusCode = "cmd_acquired" OR
	                    "DB_RobotMissionStatus".StatusCode = "cmd_executing" THEN
	                    #Dispatcher["_master"] := 1602;
	                ELSIF "DB_RobotMissionStatus".StatusCode = "cmd_rejected" OR
	                    "DB_RobotMissionStatus".StatusCode = "cmd_aborted" THEN
	                    // il robot non ha accettato: chiudi invece di restare appeso
	                    "DB_RobotMission".Command := 0;
	                    #Error := 22;
	                    #MissionCode := 0;
	                    #Dispatcher["_master"] := 0;
	                END_IF;
	            1602:
	                IF "DB_RobotMissionStatus".StatusCode = "cmd_executed" THEN
	                    "DB_RobotMission".Command := 0;
	                    // aprire = rilasciare: il lato torna vuoto
	                    #GripperOccuped[1] := FALSE;
	                    #Dispatcher["updatePartOnRobot"] := 10 + DINT_TO_INT("EMPTY");
	                    #Dispatcher["_master"] := 1603;
	                END_IF;
	            1603:
	                IF #Dispatcher["updatePartOnRobot"] = 0 THEN
	                    #MissionCode := 0;
	                    #Dispatcher["_master"] := 0;
	                END_IF;

	                ///////////// 1620: chiusura chela lato 1 (HMI)
	            1620:
	                "DB_RobotMission".Gripper_Side := 1;
	                "DB_RobotMission".Gripper_code := #Gripper_ID[1];
	                "DB_RobotMission".Command := "CMD_RobotCloseGripper1";
	                #Dispatcher["_master"] := 1621;
	            1621:
	                IF "DB_RobotMissionStatus".StatusCode = "cmd_acquired" OR
	                    "DB_RobotMissionStatus".StatusCode = "cmd_executing" THEN
	                    #Dispatcher["_master"] := 1622;
	                END_IF;
	            1622:
	                // chiudere NON implica aver preso: il contenuto resta quello
	                // dichiarato, si aggiorna solo con il comando 35
	                IF "DB_RobotMissionStatus".StatusCode = "cmd_executed" THEN
	                    "DB_RobotMission".Command := 0;
	                    #MissionCode := 0;
	                    #Dispatcher["_master"] := 0;
	                END_IF;

	                ///////////// 1640: apertura chela lato 2 (HMI)
	            1640:
	                "DB_RobotMission".Gripper_Side := 2;
	                "DB_RobotMission".Gripper_code := #Gripper_ID[2];
	                "DB_RobotMission".Command := "CMD_RobotOpenGripper2";
	                #Dispatcher["_master"] := 1641;
	            1641:
	                IF "DB_RobotMissionStatus".StatusCode = "cmd_acquired" OR
	                    "DB_RobotMissionStatus".StatusCode = "cmd_executing" THEN
	                    #Dispatcher["_master"] := 1642;
	                END_IF;
	            1642:
	                IF "DB_RobotMissionStatus".StatusCode = "cmd_executed" THEN
	                    "DB_RobotMission".Command := 0;
	                    #GripperOccuped[2] := FALSE;
	                    #Dispatcher["updatePartOnRobot"] := 20 + DINT_TO_INT("EMPTY");
	                    #Dispatcher["_master"] := 1643;
	                END_IF;
	            1643:
	                IF #Dispatcher["updatePartOnRobot"] = 0 THEN
	                    #MissionCode := 0;
	                    #Dispatcher["_master"] := 0;
	                END_IF;

